// TwinCAT 3 PLC project PLC_CRIX_VAC
// Title: plc-crix-vac
// Company: SLAC - LCLS
// ProjectVersion: 0.0.0
// ProgramVersion: 3.1.4022.7
// libraries:
//   LCLS General, * (SLAC)
//   LCLS Vacuum, * (SLAC - LCLS)
//   LCLSVacuumSerialDriverLib, * (SLAC - LCLS)
//   PMPS, * (SLAC - LCLS)
//   Tc2_SerialCom, * (Beckhoff Automation GmbH)
//   Tc2_Standard, * (Beckhoff Automation GmbH)
//   Tc2_System, * (Beckhoff Automation GmbH)
//   Tc3_Module, * (Beckhoff Automation GmbH)
// project tree:
//   / CommTask.TcTTO, PlcTask.TcTTO
//   DUTs/ E_STATES.TcDUT
//   GVLs/ GVL_ADS_Devices.TcGVL, GVL_Chamber_Gauges.TcGVL, GVL_Chamber_Valves.TcGVL, GVL_COM.TcGVL, GVL_COM_VLS.TcGVL, GVL_LI3K2.TcGVL, GVL_Mech_Room.TcGVL, GVL_PLC_Interfaces.TcGVL, GVL_PMPS.TcGVL, GVL_Pumps.TcGVL, GVL_Recirculation.TcGVL, GVL_Vars.TcGVL, GVL_VLS.TcGVL
//   POUs/ FB_ChemRIXS_Turbo_ILK.TcPOU, F_TurboGateValve_Protection_ILK_Turbo_OFF_OK_NO_GPI_READ.TcPOU, MAIN.TcPOU, PRG_ADS_Gauges.TcPOU, PRG_ADS_Interfaces.TcPOU, PRG_Chamber_Gauges.TcPOU, PRG_Chamber_Pumps.TcPOU, PRG_Chamber_Valves.TcPOU, PRG_Com.TcPOU, PRG_COM_VLS.TcPOU, PRG_LI3K2.TcPOU, PRG_Mechanical_Room.TcPOU, PRG_MPS.TcPOU, PRG_RCC.TcPOU, PRG_VLS_Turbo.TcPOU, PRG_VLS_VACUUM.TcPOU, PRG_VLS_WINDOW.TcPOU
// real-time tasks:
//   TASK PlcTask: cycle T#10ms, priority 20, ADS port 350
//   TASK CommTask: cycle T#10ms, priority 21, ADS port 351
// I/O:
//   DEVICE Device 1 (EtherCAT), AmsNetId 172.21.140.47.2.1
//     Term 1 (EK1200) [EK1200-5000 EtherCAT Power supply (2A E-Bus)]
//       Term 47 (EL6070) [EL6070 1Ch. Licensing-Terminal]
//       Term 2 (EK1122) [EK1122 2 port EtherCAT junction]
//         Hoffman Box Vac EK1 (EK1100) [EK1100 EtherCAT Coupler (2A E-Bus)]
//           E1 (EL2794)
//           E2 (EL1088) [EL1088 8Ch. Dig. Input 24V, 3ms, negative]
//           E4 (EL6002) [EL6002 Interface 2Ch. (RS232)]
//           E5 (EL6022) [EL6022 Interface 2Ch. (RS422/485)]
//           E6 (EL6022) [EL6022 Interface 2Ch. (RS422/485)]
//           E7 (EL9410)
//           E8 (EL3174) [EL3174 4Ch. Ana. Input +/-10V Diff., +/-20mA SingleEnded, 16 Bit]
//           E11 (EL3174) [EL3174 4Ch. Ana. Input +/-10V Diff., +/-20mA SingleEnded, 16 Bit]
//           E14 (EL3174) [EL3174 4Ch. Ana. Input +/-10V Diff., +/-20mA SingleEnded, 16 Bit]
//           E17 (EL2624)
//           E18 (EL9505)
//           E19 (EL1124) [EL1124 4Ch. Dig. Input 5V, 10µs, Sensor Power]
//           E20 (EL9410) [EL9410 E-Bus Power Supplier  (Diagnostics)]
//           E21 (EL2004)
//           E22 (EL1004) [EL1004 4Ch. Dig. Input 24V, 3ms]
//           E23 (EL1004)
//           E24 (EL2004) [EL2004 4Ch. Dig. Output 24V, 0.5A]
//           E25 (EL1004)
//           E26 (EL2004) [EL2004 4Ch. Dig. Output 24V, 0.5A]
//           E27 (EL1004) [EL1004 4Ch. Dig. Input 24V, 3ms]
//           E28 (EL2004)
//           E29 (EL1004) [EL1004 4Ch. Dig. Input 24V, 3ms]
//           E30 (EL2004)
//           E31 (EL1004)
//           E32 (EL9410) [EL9410 E-Bus Power Supplier  (Diagnostics)]
//           E33 (EL1004) [EL1004 4Ch. Dig. Input 24V, 3ms]
//           E34 (EL2004) [EL2004 4Ch. Dig. Output 24V, 0.5A]
//           E35 (EL1004) [EL1004 4Ch. Dig. Input 24V, 3ms]
//           E36 (EL2004)
//           E37 (EL1004)
//           E38 (EL1004) [EL1004 4Ch. Dig. Input 24V, 3ms]
//           E39 (EL2004) [EL2004 4Ch. Dig. Output 24V, 0.5A]
//           E40 (EL1004)
//           E41 (EL1004) [EL1004 4Ch. Dig. Input 24V, 3ms]
//           E42 (EL1004) [EL1004 4Ch. Dig. Input 24V, 3ms]
//           E43 (EL2794) [EL2794 4Ch. Dig. Output 24V AC/DC, 2A, short-circuit-proof]
//           E44 (EL1088) [EL1088 8Ch. Dig. Input 24V, 3ms, negative]
//           E46 (EL1004) [EL1004 4Ch. Dig. Input 24V, 3ms]
//           E47 (EL2004) [EL2004 4Ch. Dig. Output 24V, 0.5A]
//           E48 (EL9410) [EL9410 E-Bus Power Supplier  (Diagnostics)]
//           E49 (EL1004) [EL1004 4Ch. Dig. Input 24V, 3ms]
//           E50 (EL2004) [EL2004 4Ch. Dig. Output 24V, 0.5A]
//           E51 (EL4134) [EL4134 4Ch. Ana. Output -10/+10V, 16bit]
//           VLS_RCC (EK1122) [EK1122 2 port EtherCAT junction]
//             VLS_EP1 (EP6002-0002)
//             VLS_EP2 (EP2338-0001)
//             VLS_EP3 (EP2339-0021) [EP2339-0021 16 Ch. Dig. Input/Output 24V, 0,5A, M8]
//             VLS_EP4 (EP2624-0002) [EP2624-0002 4Ch. Relay Output, NO (125V AC / 30V DC)]
//             VLS_EP5 (EP3174-0002)
//             RCC_EK0 (EK1100) [EK1100 EtherCAT Coupler (2A E-Bus)]
//               RCC_E1 (EL1004) [EL1004 4Ch. Dig. Input 24V, 3ms]
//               RCC_E2 (EL2004) [EL2004 4Ch. Dig. Output 24V, 0.5A]
//               RCC_E3 (EL1004)
//               RCC_E4 (EL1004) [EL1004 4Ch. Dig. Input 24V, 3ms]
//               RCC_E5 (EL2004) [EL2004 4Ch. Dig. Output 24V, 0.5A]
//               RCC_E6 (EL1004) [EL1004 4Ch. Dig. Input 24V, 3ms]
//               RCC_E7 (EL3314) [EL3314 4Ch. Ana. Input Thermocouple (TC)]
//               RCC_E8 (EL2794) [EL2794 4Ch. Dig. Output 24V AC/DC, 2A, short-circuit-proof]
//               RCC_E9 (EL9505) [EL9505 Power supply terminal 5V]
//               RCC_E10 (EL1124)
//               Term 143 (EL3174-0002) [EL3174-0002 4Ch. Ana. Input +/-10V, +/-20mA 16 Bit, Isolated Channels]
//               RCC_E11 (EL9011)
//             RCC_GPI (901P)
//           Term 145 (EK1122) [EK1122 2 port EtherCAT junction]
//             SVLS_PR01 E0 (EK1100) [EK1100 EtherCAT Coupler (2A E-Bus)]
//               SVLS_PR01 E1 (EL6070) [EL6070 1Ch. Licensing-Terminal]
//               SVLS_PR01 E2 (EL1004) [EL1004 4Ch. Dig. Input 24V, 3ms]
//               SVLS_PR01 E3 (EL2794) [EL2794 4Ch. Dig. Output 24V AC/DC, 2A, short-circuit-proof]
//               SVLS_PR01 E4 (EL6021) [EL6021 Interface (RS422/485)]
//               SVLS_PR01 E5 (EL1004) [EL1004 4Ch. Dig. Input 24V, 3ms]
//               SVLS_PR01 E6 (EL2004) [EL2004 4Ch. Dig. Output 24V, 0.5A]
//               SVLS_PR01 E9 (EL3174-0002) [EL3174-0002 4Ch. Ana. Input +/-10V, +/-20mA 16 Bit, Isolated Channels]
//               SVLS_PR01 E10 (EL9505) [EL9505 Power supply terminal 5V]
//               SVLS_PR01 E11 (EL1124) [EL1124 4Ch. Dig. Input 5V, 10µs, Sensor Power]
//               SVLS_PR01 E12 (EL6695) [EL6695 EtherCAT Bridge terminal (Primary)]
//               SVLS_PR01 E13 (EL9011) [EL9011 End Terminal]
//           E53 (EL9011)
//         Mech Room Vac EK1 (EK1101) [EK1101 EtherCAT Coupler (2A E-Bus, ID switch)]
//           Term 45 (EL2794) [EL2794 4Ch. Dig. Output 24V AC/DC, 2A, short-circuit-proof]
//           Term 83 (EL1088) [EL1088 8Ch. Dig. Input 24V, 3ms, negative]
//           Term 92 (EL3174) [EL3174 4Ch. Ana. Input +/-10V Diff., +/-20mA SingleEnded, 16 Bit]
//           Term 93 (EL1004) [EL1004 4Ch. Dig. Input 24V, 3ms]
//           Term 94 (EL2004) [EL2004 4Ch. Dig. Output 24V, 0.5A]
//           Term 153 (EL2212) [EL2212 2Ch. dig. output with overexcitation (24V DC, 2.5A, 10A Peak)]
//           Term 96 (EL9011) [EL9011 End Terminal]
//       Term 95 (EL6695) [EL6695 EtherCAT Bridge terminal (Primary)]
//       Term 113 (EK1521-0010) [EK1521-0010 1 port EtherCAT junction (FX-SingleMode)]
//         Term 154 (EK1501-0010) [EK1501-0010 EtherCAT Coupler (2A E-Bus, FX-SingleMode, ID switch)]
//           PMPS_FFO [EL2202 2Ch. Dig. Output 24V, 0.5A]
//           PMPS_PRE [EL6695 EtherCAT Bridge terminal (Primary)]
//           Term 159 (EL9011)
// variable links:
//   PLC_CRIX_VAC Instance <-> Device 1 (EtherCAT)/Term 1 (EK1200)/Term 113 (EK1521-0010)/Term 154 (EK1501-0010)/PMPS_FFO
//     PlcTask Outputs/GVL_PMPS.g_FastFaultOutput1.q_xFastFaultOut <-> Channel 1/Output
//   PLC_CRIX_VAC Instance <-> Device 1 (EtherCAT)/Term 1 (EK1200)/Term 113 (EK1521-0010)/Term 154 (EK1501-0010)/PMPS_PRE
//     PlcTask Inputs/PRG_MPS.fbArbiterIO.i_stCurrentBP <-> IO Inputs/CurrentBP
//     PlcTask Inputs/PRG_MPS.fbArbiterIO.xTxPDO_state <-> SYNC Inputs/TxPDO state
//     PlcTask Inputs/PRG_MPS.fbArbiterIO.xTxPDO_toggle <-> SYNC Inputs/TxPDO toggle
//     PlcTask Outputs/PRG_MPS.fbArbiterIO.q_stRequestedBP <-> IO Outputs/RequestedBP
//   PLC_CRIX_VAC Instance <-> Device 1 (EtherCAT)/Term 1 (EK1200)/Term 2 (EK1122)/Hoffman Box Vac EK1 (EK1100)/E11 (EL3174)
//     PlcTask Inputs/GVL_Chamber_Gauges.CRYO_GCP_01.i_iPRESS_R <-> AI Standard Channel 2/Value
//     PlcTask Inputs/GVL_Chamber_Gauges.CRYO_GCP_02.i_iPRESS_R <-> AI Standard Channel 1/Value
//     PlcTask Inputs/GVL_Chamber_Gauges.ROUGH_GPI_01.i_iPRESS_R <-> AI Standard Channel 4/Value
//     PlcTask Inputs/GVL_Chamber_Gauges.SDS_GCP_01.i_iPRESS_R <-> AI Standard Channel 3/Value
//   PLC_CRIX_VAC Instance <-> Device 1 (EtherCAT)/Term 1 (EK1200)/Term 2 (EK1122)/Hoffman Box Vac EK1 (EK1100)/E14 (EL3174)
//     PlcTask Inputs/GVL_Chamber_Gauges.TC_GCC_01.i_iPRESS_R <-> AI Standard Channel 1/Value
//   PLC_CRIX_VAC Instance <-> Device 1 (EtherCAT)/Term 1 (EK1200)/Term 2 (EK1122)/Hoffman Box Vac EK1 (EK1100)/E17 (EL2624)
//     PlcTask Outputs/GVL_Chamber_Gauges.TC_GCC_01.q_xHV_DIS <-> Channel 1/Output
//   PLC_CRIX_VAC Instance <-> Device 1 (EtherCAT)/Term 1 (EK1200)/Term 2 (EK1122)/Hoffman Box Vac EK1 (EK1100)/E19 (EL1124)
//     PlcTask Inputs/GVL_Chamber_Gauges.TC_GCC_01.i_xDisc_Active <-> Channel 2/Input
//     PlcTask Inputs/GVL_Chamber_Gauges.TC_GCC_01.i_xHV_ON <-> Channel 1/Input
//   PLC_CRIX_VAC Instance <-> Device 1 (EtherCAT)/Term 1 (EK1200)/Term 2 (EK1122)/Hoffman Box Vac EK1 (EK1100)/E21 (EL2004)
//     PlcTask Outputs/GVL_Chamber_Valves.TC_VRC_01.q_xOPN_DO <-> Channel 1/Output
//     PlcTask Outputs/GVL_Chamber_Valves.TC_VRC_02.q_xOPN_DO <-> Channel 2/Output
//     PlcTask Outputs/GVL_Chamber_Valves.TC_VRC_03.q_xOPN_DO <-> Channel 3/Output
//     PlcTask Outputs/GVL_Chamber_Valves.VLS_VRC_01.q_xOPN_DO <-> Channel 4/Output
//   PLC_CRIX_VAC Instance <-> Device 1 (EtherCAT)/Term 1 (EK1200)/Term 2 (EK1122)/Hoffman Box Vac EK1 (EK1100)/E22 (EL1004)
//     PlcTask Inputs/GVL_Chamber_Valves.TC_VRC_01.i_xClsLS <-> Channel 2/Input
//     PlcTask Inputs/GVL_Chamber_Valves.TC_VRC_02.i_xClsLS <-> Channel 4/Input
//     PlcTask Inputs/GVL_Chamber_Valves.TC_VRC_01.i_xOpnLS <-> Channel 1/Input
//     PlcTask Inputs/GVL_Chamber_Valves.TC_VRC_02.i_xOpnLS <-> Channel 3/Input
//   PLC_CRIX_VAC Instance <-> Device 1 (EtherCAT)/Term 1 (EK1200)/Term 2 (EK1122)/Hoffman Box Vac EK1 (EK1100)/E23 (EL1004)
//     PlcTask Inputs/GVL_Chamber_Valves.TC_VRC_03.i_xClsLS <-> Channel 2/Input
//     PlcTask Inputs/GVL_Chamber_Valves.TC_VRC_03.i_xOpnLS <-> Channel 1/Input
//     PlcTask Inputs/GVL_Chamber_Valves.VLS_VRC_01.i_xClsLS <-> Channel 4/Input
//     PlcTask Inputs/GVL_Chamber_Valves.VLS_VRC_01.i_xOpnLS <-> Channel 3/Input
//   PLC_CRIX_VAC Instance <-> Device 1 (EtherCAT)/Term 1 (EK1200)/Term 2 (EK1122)/Hoffman Box Vac EK1 (EK1100)/E24 (EL2004)
//     PlcTask Outputs/GVL_Chamber_Valves.MAIN_VGC_01.q_xOPN_DO <-> Channel 3/Output
//     PlcTask Outputs/GVL_Chamber_Valves.SDS_VRC_01.q_xOPN_DO <-> Channel 1/Output
//     PlcTask Outputs/GVL_Chamber_Valves.SDS_VRC_03.q_xOPN_DO <-> Channel 2/Output
//   PLC_CRIX_VAC Instance <-> Device 1 (EtherCAT)/Term 1 (EK1200)/Term 2 (EK1122)/Hoffman Box Vac EK1 (EK1100)/E25 (EL1004)
//     PlcTask Inputs/GVL_Chamber_Valves.SDS_VRC_01.i_xClsLS <-> Channel 2/Input
//     PlcTask Inputs/GVL_Chamber_Valves.SDS_VRC_03.i_xClsLS <-> Channel 4/Input
//     PlcTask Inputs/GVL_Chamber_Valves.SDS_VRC_01.i_xOpnLS <-> Channel 1/Input
//     PlcTask Inputs/GVL_Chamber_Valves.SDS_VRC_03.i_xOpnLS <-> Channel 3/Input
//   PLC_CRIX_VAC Instance <-> Device 1 (EtherCAT)/Term 1 (EK1200)/Term 2 (EK1122)/Hoffman Box Vac EK1 (EK1100)/E26 (EL2004)
//     PlcTask Outputs/GVL_Chamber_Valves.CRYO_VGC_01.q_xCLS_DO <-> Channel 3/Output
//     PlcTask Outputs/GVL_Chamber_Valves.CRYO_VGC_01.q_xOPN_DO <-> Channel 2/Output
//     PlcTask Outputs/GVL_Chamber_Valves.CRYO_VGC_02.q_xOPN_DO <-> Channel 4/Output
//     PlcTask Outputs/GVL_Chamber_Valves.MAIN_VGC_02.q_xOPN_DO <-> Channel 1/Output
//   PLC_CRIX_VAC Instance <-> Device 1 (EtherCAT)/Term 1 (EK1200)/Term 2 (EK1122)/Hoffman Box Vac EK1 (EK1100)/E27 (EL1004)
//     PlcTask Inputs/GVL_Chamber_Valves.MAIN_VGC_01.i_xClsLS <-> Channel 2/Input
//     PlcTask Inputs/GVL_Chamber_Valves.MAIN_VGC_01.i_xOpnLS <-> Channel 1/Input
//   PLC_CRIX_VAC Instance <-> Device 1 (EtherCAT)/Term 1 (EK1200)/Term 2 (EK1122)/Hoffman Box Vac EK1 (EK1100)/E28 (EL2004)
//     PlcTask Outputs/GVL_Chamber_Valves.CRYO_VGC_02.q_xCLS_DO <-> Channel 1/Output
//     PlcTask Outputs/GVL_Chamber_Valves.CRYO_VRC_01.q_xOPN_DO <-> Channel 2/Output
//     PlcTask Outputs/GVL_Chamber_Valves.CRYO_VRC_02.q_xOPN_DO <-> Channel 3/Output
//     PlcTask Outputs/GVL_Chamber_Valves.SDS_VGC_01.q_xOPN_DO <-> Channel 4/Output
//   PLC_CRIX_VAC Instance <-> Device 1 (EtherCAT)/Term 1 (EK1200)/Term 2 (EK1122)/Hoffman Box Vac EK1 (EK1100)/E29 (EL1004)
//     PlcTask Inputs/GVL_Chamber_Valves.MAIN_VGC_02.i_xClsLS <-> Channel 1/Input
//     PlcTask Inputs/GVL_Chamber_Valves.MAIN_VGC_02.i_xOpnLS <-> Channel 2/Input
//   PLC_CRIX_VAC Instance <-> Device 1 (EtherCAT)/Term 1 (EK1200)/Term 2 (EK1122)/Hoffman Box Vac EK1 (EK1100)/E30 (EL2004)
//     PlcTask Outputs/GVL_Chamber_Valves.SDS_VGC_01.q_xCLS_DO <-> Channel 1/Output
//     PlcTask Outputs/GVL_Chamber_Valves.SDS_VRC_02.q_xOPN_DO <-> Channel 2/Output
//   PLC_CRIX_VAC Instance <-> Device 1 (EtherCAT)/Term 1 (EK1200)/Term 2 (EK1122)/Hoffman Box Vac EK1 (EK1100)/E31 (EL1004)
//     PlcTask Inputs/GVL_Chamber_Valves.CRYO_VGC_01.i_xClsLS <-> Channel 2/Input
//     PlcTask Inputs/GVL_Chamber_Valves.CRYO_VGC_01.i_xOpnLS <-> Channel 1/Input
//     PlcTask Inputs/GVL_Chamber_Valves.CRYO_VRC_01.i_xClsLS <-> Channel 4/Input
//     PlcTask Inputs/GVL_Chamber_Valves.CRYO_VRC_01.i_xOpnLS <-> Channel 3/Input
//   PLC_CRIX_VAC Instance <-> Device 1 (EtherCAT)/Term 1 (EK1200)/Term 2 (EK1122)/Hoffman Box Vac EK1 (EK1100)/E33 (EL1004)
//     PlcTask Inputs/GVL_Chamber_Valves.CRYO_VGC_02.i_xClsLS <-> Channel 2/Input
//     PlcTask Inputs/GVL_Chamber_Valves.CRYO_VGC_02.i_xOpnLS <-> Channel 1/Input
//     PlcTask Inputs/GVL_Chamber_Valves.CRYO_VRC_02.i_xClsLS <-> Channel 4/Input
//     PlcTask Inputs/GVL_Chamber_Valves.CRYO_VRC_02.i_xOpnLS <-> Channel 3/Input
//   PLC_CRIX_VAC Instance <-> Device 1 (EtherCAT)/Term 1 (EK1200)/Term 2 (EK1122)/Hoffman Box Vac EK1 (EK1100)/E35 (EL1004)
//     PlcTask Inputs/GVL_Chamber_Valves.SDS_VGC_01.i_xClsLS <-> Channel 2/Input
//     PlcTask Inputs/GVL_Chamber_Valves.SDS_VGC_01.i_xOpnLS <-> Channel 1/Input
//   PLC_CRIX_VAC Instance <-> Device 1 (EtherCAT)/Term 1 (EK1200)/Term 2 (EK1122)/Hoffman Box Vac EK1 (EK1100)/E37 (EL1004)
//     PlcTask Inputs/GVL_Chamber_Valves.SDS_VRC_02.i_xClsLS <-> Channel 2/Input
//     PlcTask Inputs/GVL_Chamber_Valves.SDS_VRC_02.i_xOpnLS <-> Channel 1/Input
//   PLC_CRIX_VAC Instance <-> Device 1 (EtherCAT)/Term 1 (EK1200)/Term 2 (EK1122)/Hoffman Box Vac EK1 (EK1100)/E39 (EL2004)
//     PlcTask Outputs/GVL_Chamber_Valves.CRIX_SVLS_VRC_01.q_xOPN_DO <-> Channel 3/Output
//     PlcTask Outputs/GVL_Chamber_Valves.SDS_VVC_01.q_xOPN_DO <-> Channel 1/Output
//     PlcTask Outputs/GVL_Chamber_Valves.SDS_VVC_02.q_xOPN_DO <-> Channel 2/Output
//   PLC_CRIX_VAC Instance <-> Device 1 (EtherCAT)/Term 1 (EK1200)/Term 2 (EK1122)/Hoffman Box Vac EK1 (EK1100)/E40 (EL1004)
//     PlcTask Inputs/GVL_Chamber_Valves.SDS_VVC_01.i_xClsLS <-> Channel 3/Input
//     PlcTask Inputs/GVL_Chamber_Valves.SDS_VVC_02.i_xClsLS <-> Channel 4/Input
//   PLC_CRIX_VAC Instance <-> Device 1 (EtherCAT)/Term 1 (EK1200)/Term 2 (EK1122)/Hoffman Box Vac EK1 (EK1100)/E41 (EL1004)
//     PlcTask Inputs/GVL_Chamber_Valves.CRIX_SVLS_VRC_01.i_xClsLS <-> Channel 2/Input
//     PlcTask Inputs/GVL_Chamber_Valves.CRIX_SVLS_VRC_01.i_xOpnLS <-> Channel 1/Input
//   PLC_CRIX_VAC Instance <-> Device 1 (EtherCAT)/Term 1 (EK1200)/Term 2 (EK1122)/Hoffman Box Vac EK1 (EK1100)/E42 (EL1004)
//     PlcTask Inputs/GVL_Pumps.TC_PTM_01.i_xAtSpd <-> Channel 4/Input
//     PlcTask Inputs/GVL_Pumps.TC_PTM_02.i_xAtSpd <-> Channel 2/Input
//     PlcTask Inputs/GVL_Pumps.TC_PTM_01.i_xFaultNC <-> Channel 3/Input
//     PlcTask Inputs/GVL_Pumps.TC_PTM_02.i_xFaultNC <-> Channel 1/Input
//   PLC_CRIX_VAC Instance <-> Device 1 (EtherCAT)/Term 1 (EK1200)/Term 2 (EK1122)/Hoffman Box Vac EK1 (EK1100)/E43 (EL2794)
//     PlcTask Outputs/GVL_Pumps.TC_PTM_01.q_RunDO <-> Channel 4/Output
//     PlcTask Outputs/GVL_Pumps.TC_PTM_02.q_RunDO <-> Channel 3/Output
//   PLC_CRIX_VAC Instance <-> Device 1 (EtherCAT)/Term 1 (EK1200)/Term 2 (EK1122)/Hoffman Box Vac EK1 (EK1100)/E46 (EL1004)
//     PlcTask Inputs/GVL_Pumps.TC_PTM_03.i_xAtSpd <-> Channel 1/Input
//     PlcTask Inputs/GVL_Pumps.TC_PTM_03.i_xFaultNC <-> Channel 3/Input
//     PlcTask Inputs/GVL_Pumps.TC_PTM_03.i_xRemote <-> Channel 2/Input
//   PLC_CRIX_VAC Instance <-> Device 1 (EtherCAT)/Term 1 (EK1200)/Term 2 (EK1122)/Hoffman Box Vac EK1 (EK1100)/E47 (EL2004)
//     PlcTask Outputs/GVL_Pumps.TC_PTM_03.q_PumpingStation <-> Channel 3/Output
//     PlcTask Outputs/GVL_Pumps.TC_PTM_03.q_RunDO <-> Channel 1/Output
//     PlcTask Outputs/GVL_Pumps.TC_PTM_03.q_xRemote <-> Channel 2/Output
//   PLC_CRIX_VAC Instance <-> Device 1 (EtherCAT)/Term 1 (EK1200)/Term 2 (EK1122)/Hoffman Box Vac EK1 (EK1100)/E49 (EL1004)
//     PlcTask Inputs/GVL_Pumps.SDS_PTM_01.i_xAtSpd <-> Channel 1/Input
//     PlcTask Inputs/GVL_Pumps.SDS_PTM_01.i_xFaultNC <-> Channel 3/Input
//     PlcTask Inputs/GVL_Pumps.SDS_PTM_01.i_xRemote <-> Channel 2/Input
//   PLC_CRIX_VAC Instance <-> Device 1 (EtherCAT)/Term 1 (EK1200)/Term 2 (EK1122)/Hoffman Box Vac EK1 (EK1100)/E5 (EL6022)
//     PlcTask Inputs/GVL_COM.K2S17_E5_CH1_stComIn/D[0] <-> COM Inputs Channel 1/Data In 0
//     PlcTask Inputs/GVL_COM.K2S17_E5_CH1_stComIn/D[10] <-> COM Inputs Channel 1/Data In 10
//     PlcTask Inputs/GVL_COM.K2S17_E5_CH1_stComIn/D[11] <-> COM Inputs Channel 1/Data In 11
//     PlcTask Inputs/GVL_COM.K2S17_E5_CH1_stComIn/D[12] <-> COM Inputs Channel 1/Data In 12
//     PlcTask Inputs/GVL_COM.K2S17_E5_CH1_stComIn/D[13] <-> COM Inputs Channel 1/Data In 13
//     PlcTask Inputs/GVL_COM.K2S17_E5_CH1_stComIn/D[14] <-> COM Inputs Channel 1/Data In 14
//     PlcTask Inputs/GVL_COM.K2S17_E5_CH1_stComIn/D[15] <-> COM Inputs Channel 1/Data In 15
//     PlcTask Inputs/GVL_COM.K2S17_E5_CH1_stComIn/D[16] <-> COM Inputs Channel 1/Data In 16
//     PlcTask Inputs/GVL_COM.K2S17_E5_CH1_stComIn/D[17] <-> COM Inputs Channel 1/Data In 17
//     PlcTask Inputs/GVL_COM.K2S17_E5_CH1_stComIn/D[18] <-> COM Inputs Channel 1/Data In 18
//     PlcTask Inputs/GVL_COM.K2S17_E5_CH1_stComIn/D[19] <-> COM Inputs Channel 1/Data In 19
//     PlcTask Inputs/GVL_COM.K2S17_E5_CH1_stComIn/D[1] <-> COM Inputs Channel 1/Data In 1
//     PlcTask Inputs/GVL_COM.K2S17_E5_CH1_stComIn/D[20] <-> COM Inputs Channel 1/Data In 20
//     PlcTask Inputs/GVL_COM.K2S17_E5_CH1_stComIn/D[21] <-> COM Inputs Channel 1/Data In 21
//     PlcTask Inputs/GVL_COM.K2S17_E5_CH1_stComIn/D[2] <-> COM Inputs Channel 1/Data In 2
//     PlcTask Inputs/GVL_COM.K2S17_E5_CH1_stComIn/D[3] <-> COM Inputs Channel 1/Data In 3
//     PlcTask Inputs/GVL_COM.K2S17_E5_CH1_stComIn/D[4] <-> COM Inputs Channel 1/Data In 4
//     PlcTask Inputs/GVL_COM.K2S17_E5_CH1_stComIn/D[5] <-> COM Inputs Channel 1/Data In 5
//     PlcTask Inputs/GVL_COM.K2S17_E5_CH1_stComIn/D[6] <-> COM Inputs Channel 1/Data In 6
//     PlcTask Inputs/GVL_COM.K2S17_E5_CH1_stComIn/D[7] <-> COM Inputs Channel 1/Data In 7
//     PlcTask Inputs/GVL_COM.K2S17_E5_CH1_stComIn/D[8] <-> COM Inputs Channel 1/Data In 8
//     PlcTask Inputs/GVL_COM.K2S17_E5_CH1_stComIn/D[9] <-> COM Inputs Channel 1/Data In 9
//     PlcTask Inputs/GVL_COM.K2S17_E5_CH2_stComIn/D[0] <-> COM Inputs Channel 2/Data In 0
//     PlcTask Inputs/GVL_COM.K2S17_E5_CH2_stComIn/D[10] <-> COM Inputs Channel 2/Data In 10
//     PlcTask Inputs/GVL_COM.K2S17_E5_CH2_stComIn/D[11] <-> COM Inputs Channel 2/Data In 11
//     PlcTask Inputs/GVL_COM.K2S17_E5_CH2_stComIn/D[12] <-> COM Inputs Channel 2/Data In 12
//     PlcTask Inputs/GVL_COM.K2S17_E5_CH2_stComIn/D[13] <-> COM Inputs Channel 2/Data In 13
//     PlcTask Inputs/GVL_COM.K2S17_E5_CH2_stComIn/D[14] <-> COM Inputs Channel 2/Data In 14
//     PlcTask Inputs/GVL_COM.K2S17_E5_CH2_stComIn/D[15] <-> COM Inputs Channel 2/Data In 15
//     PlcTask Inputs/GVL_COM.K2S17_E5_CH2_stComIn/D[16] <-> COM Inputs Channel 2/Data In 16
//     PlcTask Inputs/GVL_COM.K2S17_E5_CH2_stComIn/D[17] <-> COM Inputs Channel 2/Data In 17
//     PlcTask Inputs/GVL_COM.K2S17_E5_CH2_stComIn/D[18] <-> COM Inputs Channel 2/Data In 18
//     PlcTask Inputs/GVL_COM.K2S17_E5_CH2_stComIn/D[19] <-> COM Inputs Channel 2/Data In 19
//     PlcTask Inputs/GVL_COM.K2S17_E5_CH2_stComIn/D[1] <-> COM Inputs Channel 2/Data In 1
//     PlcTask Inputs/GVL_COM.K2S17_E5_CH2_stComIn/D[20] <-> COM Inputs Channel 2/Data In 20
//     PlcTask Inputs/GVL_COM.K2S17_E5_CH2_stComIn/D[21] <-> COM Inputs Channel 2/Data In 21
//     PlcTask Inputs/GVL_COM.K2S17_E5_CH2_stComIn/D[2] <-> COM Inputs Channel 2/Data In 2
//     PlcTask Inputs/GVL_COM.K2S17_E5_CH2_stComIn/D[3] <-> COM Inputs Channel 2/Data In 3
//     PlcTask Inputs/GVL_COM.K2S17_E5_CH2_stComIn/D[4] <-> COM Inputs Channel 2/Data In 4
//     PlcTask Inputs/GVL_COM.K2S17_E5_CH2_stComIn/D[5] <-> COM Inputs Channel 2/Data In 5
//     PlcTask Inputs/GVL_COM.K2S17_E5_CH2_stComIn/D[6] <-> COM Inputs Channel 2/Data In 6
//     PlcTask Inputs/GVL_COM.K2S17_E5_CH2_stComIn/D[7] <-> COM Inputs Channel 2/Data In 7
//     PlcTask Inputs/GVL_COM.K2S17_E5_CH2_stComIn/D[8] <-> COM Inputs Channel 2/Data In 8
//     PlcTask Inputs/GVL_COM.K2S17_E5_CH2_stComIn/D[9] <-> COM Inputs Channel 2/Data In 9
//     PlcTask Inputs/GVL_COM.K2S17_E5_CH1_stComIn/Status <-> COM Inputs Channel 1/Status
//     PlcTask Inputs/GVL_COM.K2S17_E5_CH2_stComIn/Status <-> COM Inputs Channel 2/Status
//     PlcTask Outputs/GVL_COM.K2S17_E5_CH1_stComOut/Ctrl <-> COM Outputs Channel 1/Ctrl
//     PlcTask Outputs/GVL_COM.K2S17_E5_CH2_stComOut/Ctrl <-> COM Outputs Channel 2/Ctrl
//     PlcTask Outputs/GVL_COM.K2S17_E5_CH1_stComOut/D[0] <-> COM Outputs Channel 1/Data Out 0
//     PlcTask Outputs/GVL_COM.K2S17_E5_CH1_stComOut/D[10] <-> COM Outputs Channel 1/Data Out 10
//     PlcTask Outputs/GVL_COM.K2S17_E5_CH1_stComOut/D[11] <-> COM Outputs Channel 1/Data Out 11
//     PlcTask Outputs/GVL_COM.K2S17_E5_CH1_stComOut/D[12] <-> COM Outputs Channel 1/Data Out 12
//     PlcTask Outputs/GVL_COM.K2S17_E5_CH1_stComOut/D[13] <-> COM Outputs Channel 1/Data Out 13
//     PlcTask Outputs/GVL_COM.K2S17_E5_CH1_stComOut/D[14] <-> COM Outputs Channel 1/Data Out 14
//     PlcTask Outputs/GVL_COM.K2S17_E5_CH1_stComOut/D[15] <-> COM Outputs Channel 1/Data Out 15
//     PlcTask Outputs/GVL_COM.K2S17_E5_CH1_stComOut/D[16] <-> COM Outputs Channel 1/Data Out 16
//     PlcTask Outputs/GVL_COM.K2S17_E5_CH1_stComOut/D[17] <-> COM Outputs Channel 1/Data Out 17
//     PlcTask Outputs/GVL_COM.K2S17_E5_CH1_stComOut/D[18] <-> COM Outputs Channel 1/Data Out 18
//     PlcTask Outputs/GVL_COM.K2S17_E5_CH1_stComOut/D[19] <-> COM Outputs Channel 1/Data Out 19
//     PlcTask Outputs/GVL_COM.K2S17_E5_CH1_stComOut/D[1] <-> COM Outputs Channel 1/Data Out 1
//     PlcTask Outputs/GVL_COM.K2S17_E5_CH1_stComOut/D[20] <-> COM Outputs Channel 1/Data Out 20
//     PlcTask Outputs/GVL_COM.K2S17_E5_CH1_stComOut/D[21] <-> COM Outputs Channel 1/Data Out 21
//     PlcTask Outputs/GVL_COM.K2S17_E5_CH1_stComOut/D[2] <-> COM Outputs Channel 1/Data Out 2
//     PlcTask Outputs/GVL_COM.K2S17_E5_CH1_stComOut/D[3] <-> COM Outputs Channel 1/Data Out 3
//     PlcTask Outputs/GVL_COM.K2S17_E5_CH1_stComOut/D[4] <-> COM Outputs Channel 1/Data Out 4
//     PlcTask Outputs/GVL_COM.K2S17_E5_CH1_stComOut/D[5] <-> COM Outputs Channel 1/Data Out 5
//     PlcTask Outputs/GVL_COM.K2S17_E5_CH1_stComOut/D[6] <-> COM Outputs Channel 1/Data Out 6
//     PlcTask Outputs/GVL_COM.K2S17_E5_CH1_stComOut/D[7] <-> COM Outputs Channel 1/Data Out 7
//     PlcTask Outputs/GVL_COM.K2S17_E5_CH1_stComOut/D[8] <-> COM Outputs Channel 1/Data Out 8
//     PlcTask Outputs/GVL_COM.K2S17_E5_CH1_stComOut/D[9] <-> COM Outputs Channel 1/Data Out 9
//     PlcTask Outputs/GVL_COM.K2S17_E5_CH2_stComOut/D[0] <-> COM Outputs Channel 2/Data Out 0
//     PlcTask Outputs/GVL_COM.K2S17_E5_CH2_stComOut/D[10] <-> COM Outputs Channel 2/Data Out 10
//     PlcTask Outputs/GVL_COM.K2S17_E5_CH2_stComOut/D[11] <-> COM Outputs Channel 2/Data Out 11
//     PlcTask Outputs/GVL_COM.K2S17_E5_CH2_stComOut/D[12] <-> COM Outputs Channel 2/Data Out 12
//     PlcTask Outputs/GVL_COM.K2S17_E5_CH2_stComOut/D[13] <-> COM Outputs Channel 2/Data Out 13
//     PlcTask Outputs/GVL_COM.K2S17_E5_CH2_stComOut/D[14] <-> COM Outputs Channel 2/Data Out 14
//     PlcTask Outputs/GVL_COM.K2S17_E5_CH2_stComOut/D[15] <-> COM Outputs Channel 2/Data Out 15
//     PlcTask Outputs/GVL_COM.K2S17_E5_CH2_stComOut/D[16] <-> COM Outputs Channel 2/Data Out 16
//     PlcTask Outputs/GVL_COM.K2S17_E5_CH2_stComOut/D[17] <-> COM Outputs Channel 2/Data Out 17
//     PlcTask Outputs/GVL_COM.K2S17_E5_CH2_stComOut/D[18] <-> COM Outputs Channel 2/Data Out 18
//     PlcTask Outputs/GVL_COM.K2S17_E5_CH2_stComOut/D[19] <-> COM Outputs Channel 2/Data Out 19
//     PlcTask Outputs/GVL_COM.K2S17_E5_CH2_stComOut/D[1] <-> COM Outputs Channel 2/Data Out 1
//     PlcTask Outputs/GVL_COM.K2S17_E5_CH2_stComOut/D[20] <-> COM Outputs Channel 2/Data Out 20
//     PlcTask Outputs/GVL_COM.K2S17_E5_CH2_stComOut/D[21] <-> COM Outputs Channel 2/Data Out 21
//     PlcTask Outputs/GVL_COM.K2S17_E5_CH2_stComOut/D[2] <-> COM Outputs Channel 2/Data Out 2
//     PlcTask Outputs/GVL_COM.K2S17_E5_CH2_stComOut/D[3] <-> COM Outputs Channel 2/Data Out 3
//     PlcTask Outputs/GVL_COM.K2S17_E5_CH2_stComOut/D[4] <-> COM Outputs Channel 2/Data Out 4
//     PlcTask Outputs/GVL_COM.K2S17_E5_CH2_stComOut/D[5] <-> COM Outputs Channel 2/Data Out 5
//     PlcTask Outputs/GVL_COM.K2S17_E5_CH2_stComOut/D[6] <-> COM Outputs Channel 2/Data Out 6
//     PlcTask Outputs/GVL_COM.K2S17_E5_CH2_stComOut/D[7] <-> COM Outputs Channel 2/Data Out 7
//     PlcTask Outputs/GVL_COM.K2S17_E5_CH2_stComOut/D[8] <-> COM Outputs Channel 2/Data Out 8
//     PlcTask Outputs/GVL_COM.K2S17_E5_CH2_stComOut/D[9] <-> COM Outputs Channel 2/Data Out 9
//   PLC_CRIX_VAC Instance <-> Device 1 (EtherCAT)/Term 1 (EK1200)/Term 2 (EK1122)/Hoffman Box Vac EK1 (EK1100)/E50 (EL2004)
//     PlcTask Outputs/GVL_Pumps.SDS_PTM_01.q_PumpingStation <-> Channel 3/Output
//     PlcTask Outputs/GVL_Pumps.SDS_PTM_01.q_RunDO <-> Channel 1/Output
//     PlcTask Outputs/GVL_Pumps.SDS_PTM_01.q_xRemote <-> Channel 2/Output
//   PLC_CRIX_VAC Instance <-> Device 1 (EtherCAT)/Term 1 (EK1200)/Term 2 (EK1122)/Hoffman Box Vac EK1 (EK1100)/E8 (EL3174)
//     PlcTask Inputs/GVL_Chamber_Gauges.CRYO_GPI_01.i_iPRESS_R <-> AI Standard Channel 3/Value
//     PlcTask Inputs/GVL_Chamber_Gauges.TC_GCP_01.i_iPRESS_R <-> AI Standard Channel 4/Value
//     PlcTask Inputs/GVL_Chamber_Gauges.TC_GPI_01.i_iPRESS_R <-> AI Standard Channel 2/Value
//   PLC_CRIX_VAC Instance <-> Device 1 (EtherCAT)/Term 1 (EK1200)/Term 2 (EK1122)/Hoffman Box Vac EK1 (EK1100)/Term 145 (EK1122)/SVLS_PR01 E0 (EK1100)/SVLS_PR01 E11 (EL1124)
//     PlcTask Inputs/GVL_Pumps.CRIX_SVLS_PIP_1.i_xError <-> Channel 2/Input
//     PlcTask Inputs/GVL_Pumps.CRIX_SVLS_PIP_1.i_xIP_ON <-> Channel 1/Input
//   PLC_CRIX_VAC Instance <-> Device 1 (EtherCAT)/Term 1 (EK1200)/Term 2 (EK1122)/Hoffman Box Vac EK1 (EK1100)/Term 145 (EK1122)/SVLS_PR01 E0 (EK1100)/SVLS_PR01 E2 (EL1004)
//     PlcTask Inputs/GVL_Pumps.CRIX_SVLS_PTM_01.i_xAtSpd <-> Channel 1/Input
//     PlcTask Inputs/GVL_Pumps.CRIX_SVLS_PTM_01.i_xFaultNC <-> Channel 2/Input
//   PLC_CRIX_VAC Instance <-> Device 1 (EtherCAT)/Term 1 (EK1200)/Term 2 (EK1122)/Hoffman Box Vac EK1 (EK1100)/Term 145 (EK1122)/SVLS_PR01 E0 (EK1100)/SVLS_PR01 E3 (EL2794)
//     PlcTask Outputs/GVL_Pumps.CRIX_SVLS_PIP_1.q_xHVEna_DO <-> Channel 3/Output
//     PlcTask Outputs/GVL_Pumps.CRIX_SVLS_PTM_01.q_RunDO <-> Channel 1/Output
//     PlcTask Outputs/GVL_Pumps.CRIX_SVLS_PTM_01.q_xReset <-> Channel 2/Output
//   PLC_CRIX_VAC Instance <-> Device 1 (EtherCAT)/Term 1 (EK1200)/Term 2 (EK1122)/Hoffman Box Vac EK1 (EK1100)/Term 145 (EK1122)/SVLS_PR01 E0 (EK1100)/SVLS_PR01 E4 (EL6021)
//     PlcTask Inputs/GVL_COM.CRIX_SVLS_stComIn/D[{0..21}] <-> COM TxPDO-Map Inputs/Data In {0..21}  (22 links)
//     PlcTask Inputs/GVL_COM.CRIX_SVLS_stComIn/Status <-> COM TxPDO-Map Inputs/Status
//     PlcTask Outputs/GVL_COM.CRIX_SVLS_stComOut/Ctrl <-> COM RxPDO-Map Outputs/Ctrl
//     PlcTask Outputs/GVL_COM.CRIX_SVLS_stComOut/D[{0..21}] <-> COM RxPDO-Map Outputs/Data Out {0..21}  (22 links)
//   PLC_CRIX_VAC Instance <-> Device 1 (EtherCAT)/Term 1 (EK1200)/Term 2 (EK1122)/Hoffman Box Vac EK1 (EK1100)/Term 145 (EK1122)/SVLS_PR01 E0 (EK1100)/SVLS_PR01 E5 (EL1004)
//     PlcTask Inputs/GVL_Chamber_Valves.CRIX_SVLS_VWC_01.i_xClsLS <-> Channel 2/Input
//     PlcTask Inputs/GVL_Chamber_Valves.CRIX_SVLS_VWC_01.i_xOpnLS <-> Channel 1/Input
//   PLC_CRIX_VAC Instance <-> Device 1 (EtherCAT)/Term 1 (EK1200)/Term 2 (EK1122)/Hoffman Box Vac EK1 (EK1100)/Term 145 (EK1122)/SVLS_PR01 E0 (EK1100)/SVLS_PR01 E6 (EL2004)
//     PlcTask Outputs/GVL_Chamber_Valves.CRIX_SVLS_VWC_01.q_xCLS_DO <-> Channel 1/Output
//   PLC_CRIX_VAC Instance <-> Device 1 (EtherCAT)/Term 1 (EK1200)/Term 2 (EK1122)/Hoffman Box Vac EK1 (EK1100)/Term 145 (EK1122)/SVLS_PR01 E0 (EK1100)/SVLS_PR01 E9 (EL3174-0002)
//     PlcTask Inputs/GVL_Chamber_Gauges.CRIX_SVLS_GCP_01.i_iPRESS_R <-> AI Standard Channel 1/Value
//     PlcTask Inputs/GVL_Chamber_Gauges.CRIX_SVLS_GCP_02.i_iPRESS_R <-> AI Standard Channel 2/Value
//     PlcTask Inputs/GVL_Pumps.CRIX_SVLS_PIP_1.i_iPRESS <-> AI Standard Channel 1/Value
//   PLC_CRIX_VAC Instance <-> Device 1 (EtherCAT)/Term 1 (EK1200)/Term 2 (EK1122)/Hoffman Box Vac EK1 (EK1100)/VLS_RCC (EK1122)/RCC_EK0 (EK1100)/RCC_E1 (EL1004)
//     PlcTask Inputs/GVL_Recirculation.RCC_VRC_01.i_xClsLS <-> Channel 1/Input
//     PlcTask Inputs/GVL_Recirculation.RCC_VRC_02.i_xClsLS <-> Channel 2/Input
//     PlcTask Inputs/GVL_Recirculation.RCC_VRC_03.i_xClsLS <-> Channel 3/Input
//     PlcTask Inputs/GVL_Recirculation.RCC_VRC_02.i_xOpnLS <-> Channel 4/Input
//   PLC_CRIX_VAC Instance <-> Device 1 (EtherCAT)/Term 1 (EK1200)/Term 2 (EK1122)/Hoffman Box Vac EK1 (EK1100)/VLS_RCC (EK1122)/RCC_EK0 (EK1100)/RCC_E2 (EL2004)
//     PlcTask Outputs/GVL_Recirculation.RCC_VRC_01.q_xOPN_DO <-> Channel 1/Output
//     PlcTask Outputs/GVL_Recirculation.RCC_VRC_02.q_xOPN_DO <-> Channel 2/Output
//     PlcTask Outputs/GVL_Recirculation.RCC_VRC_03.q_xOPN_DO <-> Channel 3/Output
//     PlcTask Outputs/GVL_Recirculation.RCC_VRC_04.q_xOPN_DO <-> Channel 4/Output
//   PLC_CRIX_VAC Instance <-> Device 1 (EtherCAT)/Term 1 (EK1200)/Term 2 (EK1122)/Hoffman Box Vac EK1 (EK1100)/VLS_RCC (EK1122)/RCC_EK0 (EK1100)/RCC_E3 (EL1004)
//     PlcTask Inputs/GVL_Recirculation.RCC_VRC_04.i_xClsLS <-> Channel 1/Input
//   PLC_CRIX_VAC Instance <-> Device 1 (EtherCAT)/Term 1 (EK1200)/Term 2 (EK1122)/Hoffman Box Vac EK1 (EK1100)/VLS_RCC (EK1122)/RCC_EK0 (EK1100)/RCC_E7 (EL3314)
//     PlcTask Inputs/GVL_Recirculation.RCC_STC_01.bError <-> TC Inputs Channel 3/Status/Error
//     PlcTask Inputs/GVL_Recirculation.RCC_STC_02.bError <-> TC Inputs Channel 4/Status/Error
//     PlcTask Inputs/GVL_Recirculation.RCC_STC_01.bOverrange <-> TC Inputs Channel 3/Status/Overrange
//     PlcTask Inputs/GVL_Recirculation.RCC_STC_02.bOverrange <-> TC Inputs Channel 4/Status/Overrange
//     PlcTask Inputs/GVL_Recirculation.RCC_STC_01.bUnderrange <-> TC Inputs Channel 3/Status/Underrange
//     PlcTask Inputs/GVL_Recirculation.RCC_STC_02.bUnderrange <-> TC Inputs Channel 4/Status/Underrange
//     PlcTask Inputs/GVL_Recirculation.RCC_STC_01.iRaw <-> TC Inputs Channel 3/Value
//     PlcTask Inputs/GVL_Recirculation.RCC_STC_02.iRaw <-> TC Inputs Channel 4/Value
//   PLC_CRIX_VAC Instance <-> Device 1 (EtherCAT)/Term 1 (EK1200)/Term 2 (EK1122)/Hoffman Box Vac EK1 (EK1100)/VLS_RCC (EK1122)/RCC_GPI (901P)
//     PlcTask Inputs/GVL_Recirculation.RCC_GCP_01.bWcstate <-> WcState/WcState
//     PlcTask Inputs/GVL_Recirculation.RCC_GCP_01.i_iPRESS_R <-> TXPDO Combined/Combination Gauge Active Value
//     PlcTask Inputs/GVL_Recirculation.RCC_GCP_01.xOverrange <-> TXPDO Combined/Combination Gauge Overrange Exceeded
//     PlcTask Inputs/GVL_Recirculation.RCC_GCP_01.xPress_OK <-> TXPDO Combined/Combination Gauge Reading Valid
//     PlcTask Inputs/GVL_Recirculation.RCC_GCP_01.xUnderrange <-> TXPDO Combined/Combination Gauge Underrange Exceeded
//   PLC_CRIX_VAC Instance <-> Device 1 (EtherCAT)/Term 1 (EK1200)/Term 2 (EK1122)/Hoffman Box Vac EK1 (EK1100)/VLS_RCC (EK1122)/VLS_EP1 (EP6002-0002)
//     PlcTask Inputs/GVL_COM_VLS.VLS_EP1_CH1_stComIn/D[{0..21}] <-> COM TxPDO-Map Inputs Channel 1/Data In {0..21}  (22 links)
//     PlcTask Inputs/GVL_COM_VLS.VLS_EP1_CH1_stComIn/Status <-> COM TxPDO-Map Inputs Channel 1/Status
//     PlcTask Outputs/GVL_COM_VLS.VLS_EP1_CH1_stComOut/Ctrl <-> COM RxPDO-Map Outputs Channel 1/Ctrl
//     PlcTask Outputs/GVL_COM_VLS.VLS_EP1_CH1_stComOut/D[{0..21}] <-> COM RxPDO-Map Outputs Channel 1/Data Out {0..21}  (22 links)
//   PLC_CRIX_VAC Instance <-> Device 1 (EtherCAT)/Term 1 (EK1200)/Term 2 (EK1122)/Hoffman Box Vac EK1 (EK1100)/VLS_RCC (EK1122)/VLS_EP2 (EP2338-0001)
//     PlcTask Inputs/GVL_VLS.VLS_PTM_01.i_xAtSpd <-> Channel 1/Input
//     PlcTask Inputs/GVL_VLS.VLS_PTM_01.i_xFaultNC <-> Channel 2/Input
//   PLC_CRIX_VAC Instance <-> Device 1 (EtherCAT)/Term 1 (EK1200)/Term 2 (EK1122)/Hoffman Box Vac EK1 (EK1100)/VLS_RCC (EK1122)/VLS_EP3 (EP2339-0021)
//     PlcTask Inputs/GVL_VLS.VLS_VGC_01.i_xClsLS <-> Channel 7/Input
//     PlcTask Inputs/GVL_VLS.VLS_VGC_01.i_xOpnLS <-> Channel 6/Input
//     PlcTask Inputs/GVL_VLS.VLS_VWC_01.i_xClsLS <-> Channel 10/Input
//     PlcTask Inputs/GVL_VLS.VLS_VWC_01.i_xOpnLS <-> Channel 9/Input
//     PlcTask Outputs/GVL_VLS.VLS_VGC_01.q_xOPN_DO <-> Channel 21/Output
//     PlcTask Outputs/GVL_VLS.VLS_VWC_01.q_xCLS_DO <-> Channel 24/Output
//   PLC_CRIX_VAC Instance <-> Device 1 (EtherCAT)/Term 1 (EK1200)/Term 2 (EK1122)/Hoffman Box Vac EK1 (EK1100)/VLS_RCC (EK1122)/VLS_EP4 (EP2624-0002)
//     PlcTask Outputs/GVL_VLS.VLS_GCC_01.q_xHV_DIS <-> Channel 1/Output
//     PlcTask Outputs/GVL_VLS.VLS_PTM_01.q_RunDO <-> Channel 3/Output
//   PLC_CRIX_VAC Instance <-> Device 1 (EtherCAT)/Term 1 (EK1200)/Term 2 (EK1122)/Hoffman Box Vac EK1 (EK1100)/VLS_RCC (EK1122)/VLS_EP5 (EP3174-0002)
//     PlcTask Inputs/GVL_VLS.VLS_GCC_01.i_iPRESS_R <-> AI Standard Channel 2/Value
//     PlcTask Inputs/GVL_VLS.VLS_GPI_01.i_iPRESS_R <-> AI Standard Channel 1/Value
//     PlcTask Inputs/GVL_VLS.VLS_ROUGH_GPI.i_iPRESS_R <-> AI Standard Channel 3/Value
//   PLC_CRIX_VAC Instance <-> Device 1 (EtherCAT)/Term 1 (EK1200)/Term 2 (EK1122)/Mech Room Vac EK1 (EK1101)/Term 153 (EL2212)
//     PlcTask Outputs/GVL_Mech_Room.MECH_VVC_01.q_xOPN_DO <-> DOX Control Channel 2/Control/Output
//   PLC_CRIX_VAC Instance <-> Device 1 (EtherCAT)/Term 1 (EK1200)/Term 2 (EK1122)/Mech Room Vac EK1 (EK1101)/Term 45 (EL2794)
//     PlcTask Outputs/GVL_Mech_Room.MECH_PRO_01.q_xBPStart <-> Channel 2/Output
//     PlcTask Outputs/GVL_Mech_Room.MECH_PRO_01.q_xMPStart <-> Channel 1/Output
//   PLC_CRIX_VAC Instance <-> Device 1 (EtherCAT)/Term 1 (EK1200)/Term 2 (EK1122)/Mech Room Vac EK1 (EK1101)/Term 83 (EL1088)
//     PlcTask Inputs/GVL_Mech_Room.MECH_PRO_01.i_xAlarmOK <-> Channel 4/Input
//     PlcTask Inputs/GVL_Mech_Room.MECH_PRO_01.i_xBPStatus <-> Channel 2/Input
//     PlcTask Inputs/GVL_Mech_Room.MECH_PRO_01.i_xMPStatus <-> Channel 1/Input
//     PlcTask Inputs/GVL_Mech_Room.MECH_PRO_01.i_xRemote <-> Channel 5/Input
//     PlcTask Inputs/GVL_Mech_Room.MECH_PRO_01.i_xWarning <-> Channel 3/Input
//   PLC_CRIX_VAC Instance <-> Device 1 (EtherCAT)/Term 1 (EK1200)/Term 2 (EK1122)/Mech Room Vac EK1 (EK1101)/Term 92 (EL3174)
//     PlcTask Inputs/GVL_Mech_Room.MECH_GPI_01.i_iPRESS_R <-> AI Standard Channel 1/Value
//   PLC_CRIX_VAC Instance <-> Device 1 (EtherCAT)/Term 1 (EK1200)/Term 95 (EL6695)
//     PlcTask Inputs/GVL_PLC_Interfaces.xEcatBridge_External_device_not_connected <-> SYNC Inputs/External device not connected
//     PlcTask Inputs/GVL_PLC_Interfaces.xEcatBridge_TxPDO_state <-> SYNC Inputs/TxPDO state
//     PlcTask Inputs/GVL_PLC_Interfaces.xEcatBridge_WcState <-> WcState/WcState
//     PlcTask Inputs/GVL_PLC_Interfaces.xPTC_MOT_Y_10_IN <-> IO Inputs/bMOTY10_IN
//     PlcTask Inputs/GVL_PLC_Interfaces.xPTC_MOT_Y_11_IN <-> IO Inputs/bMOTY11_IN
//     PlcTask Inputs/GVL_PLC_Interfaces.xPTC_MOT_Y_10_OUT <-> IO Inputs/bMOTY10_OUT
//     PlcTask Inputs/GVL_PLC_Interfaces.xPTC_MOT_Y_11_OUT <-> IO Inputs/bMOTY11_OUT
//     PlcTask Inputs/GVL_PLC_Interfaces.xSDS_MOT_Z_18_IN <-> IO Inputs/xSDS_MOT_Z_18_IN
//     PlcTask Inputs/GVL_PLC_Interfaces.xSDS_MOT_Z_18_OUT <-> IO Inputs/xSDS_MOT_Z_18_OUT
//     PlcTask Outputs/GVL_PLC_Interfaces.bCRYO_VGC_01_CLS <-> IO Outputs/bCRYO_VGC_01_CLS
//     PlcTask Outputs/GVL_PLC_Interfaces.bCRYO_VGC_02_CLS <-> IO Outputs/bCRYO_VGC_02_CLS
//     PlcTask Outputs/GVL_PLC_Interfaces.bCRYO_VGC_01_OPN <-> IO Outputs/bCRYO_VGC_01_OPN
//     PlcTask Outputs/GVL_PLC_Interfaces.bCRYO_VGC_02_OPN <-> IO Outputs/bCRYO_VGC_02_OPN
//     PlcTask Outputs/GVL_PLC_Interfaces.bSDS_VGC_01_CLS <-> IO Outputs/bSDS_VGC_01_CLS
//     PlcTask Outputs/GVL_PLC_Interfaces.bSDS_VGC_01_OPN <-> IO Outputs/bSDS_VGC_01_OPN

CONFIGURATION PLC_CRIX_VAC
    RESOURCE PLC ON TwinCAT3
        TASK CommTask(INTERVAL := T#10ms, PRIORITY := 21);
        TASK PlcTask(INTERVAL := T#10ms, PRIORITY := 20);
        PROGRAM PRG_COM_VLS WITH CommTask : PRG_COM_VLS;
        PROGRAM MAIN WITH PlcTask : MAIN;
    END_RESOURCE
END_CONFIGURATION

// ---- DUTs/E_STATES.TcDUT
{attribute 'qualified_only'}
{attribute 'strict'}
TYPE E_STATES :
(
    INIT := 0,
    SETUP,
    OVERRIDE,
    READY,
    NOT_SAFE
);
END_TYPE

// ---- GVLs/GVL_ADS_Devices.TcGVL
//{attribute 'qualified_only'}
VAR_GLOBAL

 {attribute 'pytmc' :=' pv: TM2K2:GCC:01:reader '}
    TM2K2_GCC_01_reader : FB_TGCC_ADS;
 {attribute 'pytmc' :=' pv: AT3K2:GCC:01:reader '}
    AT3K2_GCC_01_reader : FB_TGCC_ADS;

END_VAR

// ---- GVLs/GVL_Chamber_Gauges.TcGVL
//{attribute 'qualified_only'}
VAR_GLOBAL
    (* Pirani & Cold Cathode*)

    {attribute 'pytmc' :=' pv: CRIXS:TC:GPI:01 '}
    {attribute 'TcLinkTo' := 	'.i_iPRESS_R	:=	TIID^Device 1 (EtherCAT)^Term 1 (EK1200)^Term 2 (EK1122)^Hoffman Box Vac EK1 (EK1100)^E8 (EL3174)^AI Standard Channel 2^Value '}
    TC_GPI_01 : FB_MKS275;

    stTC_GPI_01 : ST_VG;


    {attribute 'pytmc' :=' pv: CRIXS:CRYO:GPI:01 '}
    {attribute 'TcLinkTo' := 	'.i_iPRESS_R	:=	TIID^Device 1 (EtherCAT)^Term 1 (EK1200)^Term 2 (EK1122)^Hoffman Box Vac EK1 (EK1100)^E8 (EL3174)^AI Standard Channel 3^Value '}
    CRYO_GPI_01 : FB_MKS275;

    stCRYO_GPI_01 : ST_VG;


    {attribute 'pytmc' :=' pv: CRIXS:ROUGH:GPI:01 '}
    {attribute 'TcLinkTo' := 	'.i_iPRESS_R	:=	TIID^Device 1 (EtherCAT)^Term 1 (EK1200)^Term 2 (EK1122)^Hoffman Box Vac EK1 (EK1100)^E11 (EL3174)^AI Standard Channel 4^Value '}
    ROUGH_GPI_01 : FB_MKS275;

    stROUGH_GPI_01 : ST_VG;

    {attribute 'pytmc' :=' pv: CRIXS:TC:GCC:01 '}
    {attribute 'TcLinkTo' := 	'.i_iPRESS_R	:=	TIID^Device 1 (EtherCAT)^Term 1 (EK1200)^Term 2 (EK1122)^Hoffman Box Vac EK1 (EK1100)^E14 (EL3174)^AI Standard Channel 1^Value;
                                 .i_xHV_ON	    :=	TIID^Device 1 (EtherCAT)^Term 1 (EK1200)^Term 2 (EK1122)^Hoffman Box Vac EK1 (EK1100)^E19 (EL1124)^Channel 1^Input;
                                 .i_xDisc_Active:=	TIID^Device 1 (EtherCAT)^Term 1 (EK1200)^Term 2 (EK1122)^Hoffman Box Vac EK1 (EK1100)^E19 (EL1124)^Channel 2^Input;
                                 .q_xHV_DIS		:= 	TIID^Device 1 (EtherCAT)^Term 1 (EK1200)^Term 2 (EK1122)^Hoffman Box Vac EK1 (EK1100)^E17 (EL2624)^Channel 1^Output	'}
    TC_GCC_01 : FB_MKS500;

    stTC_GCC_01 : ST_VG;

    (* Micro Pirani combination gauges *)


    {attribute 'pytmc' :=' pv: CRIXS:CRYO:GCP:01 '}
    {attribute 'TcLinkTo' := 	'.i_iPRESS_R	:= TIID^Device 1 (EtherCAT)^Term 1 (EK1200)^Term 2 (EK1122)^Hoffman Box Vac EK1 (EK1100)^E11 (EL3174)^AI Standard Channel 2^Value '}
    CRYO_GCP_01 : FB_972;

    stCRYO_GCP_01 : ST_VG;

    {attribute 'pytmc' :=' pv: CRIXS:CRYO:GCP:02 '}
    {attribute 'TcLinkTo' := 	'.i_iPRESS_R	:= TIID^Device 1 (EtherCAT)^Term 1 (EK1200)^Term 2 (EK1122)^Hoffman Box Vac EK1 (EK1100)^E11 (EL3174)^AI Standard Channel 1^Value '}
    CRYO_GCP_02 : FB_972;

    stCRYO_GCP_02 : ST_VG;

    {attribute 'pytmc' :=' pv: CRIXS:SDS:GCP:01 '}
    {attribute 'TcLinkTo' := 	'.i_iPRESS_R	:= TIID^Device 1 (EtherCAT)^Term 1 (EK1200)^Term 2 (EK1122)^Hoffman Box Vac EK1 (EK1100)^E11 (EL3174)^AI Standard Channel 3^Value '}
    SDS_GCP_01 : FB_972;

    stSDS_GCP_01 : ST_VG;

    {attribute 'pytmc' :=' pv: CRIXS:TC:GCP:01 '}
    {attribute 'TcLinkTo' := 	'.i_iPRESS_R	:=	TIID^Device 1 (EtherCAT)^Term 1 (EK1200)^Term 2 (EK1122)^Hoffman Box Vac EK1 (EK1100)^E8 (EL3174)^AI Standard Channel 4^Value '}
    TC_GCP_01 : FB_972;

    stTC_GCP_01 : ST_VG;

    {attribute 'pytmc' :=' pv: CRIXS:SVLS:GCP:01 '}
    {attribute 'TcLinkTo' := 	'.i_iPRESS_R	:=	TIIB[SVLS_PR01 E9 (EL3174-0002)]^AI Standard Channel 1^Value '}
    CRIX_SVLS_GCP_01 : FB_972;

    stCRIX_SVLS_GCP_01 : ST_VG;

    {attribute 'pytmc' :=' pv: CRIXS:SVLS:GCP:02 '}
    {attribute 'TcLinkTo' := 	'.i_iPRESS_R	:=	TIIB[SVLS_PR01 E9 (EL3174-0002)]^AI Standard Channel 2^Value '}
    CRIX_SVLS_GCP_02 : FB_972;

    stCRIX_SVLS_GCP_02 : ST_VG;

END_VAR

// ---- GVLs/GVL_Chamber_Valves.TcGVL
//{attribute 'qualified_only'}
VAR_GLOBAL

    (* Roughing Manifold Valvese *)

    (*
    {attribute 'pytmc' :=' pv: CRIX:VGC:01 '}
    {attribute 'TcLinkTo' := 	'.i_xOpnLS	:=	TIID^Device 1 (EtherCAT)^Term 1 (EK1200)^Term 2 (EK1122)^Hoffman Box Vac EK1 (EK1100)^E41 (EL1004)^Channel 1^Input;
                                 .i_xClsLS	:=	TIID^Device 1 (EtherCAT)^Term 1 (EK1200)^Term 2 (EK1122)^Hoffman Box Vac EK1 (EK1100)^E41 (EL1004)^Channel 2^Input;
                                .q_xOPN_DO	:=	TIID^Device 1 (EtherCAT)^Term 1 (EK1200)^Term 2 (EK1122)^Hoffman Box Vac EK1 (EK1100)^E39 (EL2004)^Channel 3^Output'}
    CRIX_VGC_01 : FB_VRC;

    stCRIX_VGC_01 : ST_VRC;
    *)

    {attribute 'pytmc' :=' pv: CRIXS:TC:VRC:01 '}
    {attribute 'TcLinkTo' := 	'.i_xOpnLS	:=	TIID^Device 1 (EtherCAT)^Term 1 (EK1200)^Term 2 (EK1122)^Hoffman Box Vac EK1 (EK1100)^E22 (EL1004)^Channel 1^Input;
                                 .i_xClsLS	:=	TIID^Device 1 (EtherCAT)^Term 1 (EK1200)^Term 2 (EK1122)^Hoffman Box Vac EK1 (EK1100)^E22 (EL1004)^Channel 2^Input;
                                .q_xOPN_DO	:=	TIID^Device 1 (EtherCAT)^Term 1 (EK1200)^Term 2 (EK1122)^Hoffman Box Vac EK1 (EK1100)^E21 (EL2004)^Channel 1^Output'}

    TC_VRC_01 : FB_VGC_2S;

    stTC_VRC_01 : ST_VGC_2S;

    {attribute 'pytmc' :=' pv: CRIXS:TC:VRC:02 '}
    {attribute 'TcLinkTo' := 	'.i_xOpnLS	:=	TIID^Device 1 (EtherCAT)^Term 1 (EK1200)^Term 2 (EK1122)^Hoffman Box Vac EK1 (EK1100)^E22 (EL1004)^Channel 3^Input;
                                 .i_xClsLS	:=	TIID^Device 1 (EtherCAT)^Term 1 (EK1200)^Term 2 (EK1122)^Hoffman Box Vac EK1 (EK1100)^E22 (EL1004)^Channel 4^Input;
                                .q_xOPN_DO	:=	TIID^Device 1 (EtherCAT)^Term 1 (EK1200)^Term 2 (EK1122)^Hoffman Box Vac EK1 (EK1100)^E21 (EL2004)^Channel 2^Output'}

    TC_VRC_02 : FB_VRC;

    stTC_VRC_02 : ST_VRC;

    {attribute 'pytmc' :=' pv: CRIXS:TC:VRC:03 '}
    {attribute 'TcLinkTo' := 	'.i_xOpnLS	:=	TIID^Device 1 (EtherCAT)^Term 1 (EK1200)^Term 2 (EK1122)^Hoffman Box Vac EK1 (EK1100)^E23 (EL1004)^Channel 1^Input;
                                 .i_xClsLS	:=	TIID^Device 1 (EtherCAT)^Term 1 (EK1200)^Term 2 (EK1122)^Hoffman Box Vac EK1 (EK1100)^E23 (EL1004)^Channel 2^Input;
                                .q_xOPN_DO	:=	TIID^Device 1 (EtherCAT)^Term 1 (EK1200)^Term 2 (EK1122)^Hoffman Box Vac EK1 (EK1100)^E21 (EL2004)^Channel 3^Output'}

    TC_VRC_03 : FB_VRC;
    stTC_VRC_03 : ST_VRC;


    {attribute 'pytmc' :=' pv: CRIXS:VLS:VRC:01 '}
    {attribute 'TcLinkTo' := 	'.i_xOpnLS	:=	TIID^Device 1 (EtherCAT)^Term 1 (EK1200)^Term 2 (EK1122)^Hoffman Box Vac EK1 (EK1100)^E23 (EL1004)^Channel 3^Input;
                                 .i_xClsLS	:=	TIID^Device 1 (EtherCAT)^Term 1 (EK1200)^Term 2 (EK1122)^Hoffman Box Vac EK1 (EK1100)^E23 (EL1004)^Channel 4^Input;
                                .q_xOPN_DO	:=	TIID^Device 1 (EtherCAT)^Term 1 (EK1200)^Term 2 (EK1122)^Hoffman Box Vac EK1 (EK1100)^E21 (EL2004)^Channel 4^Output'}

    VLS_VRC_01 : FB_VRC;

    stVLS_VRC_01 : ST_VRC;

    (*
    stCRIX_VGC_03 : ST_VRC;
    *)
    {attribute 'pytmc' :=' pv: CRIXS:SDS:VRC:03 '}
    {attribute 'TcLinkTo' := 	'.i_xOpnLS	:=	TIID^Device 1 (EtherCAT)^Term 1 (EK1200)^Term 2 (EK1122)^Hoffman Box Vac EK1 (EK1100)^E25 (EL1004)^Channel 3^Input;
                                 .i_xClsLS	:=	TIID^Device 1 (EtherCAT)^Term 1 (EK1200)^Term 2 (EK1122)^Hoffman Box Vac EK1 (EK1100)^E25 (EL1004)^Channel 4^Input;
                                .q_xOPN_DO	:=	TIID^Device 1 (EtherCAT)^Term 1 (EK1200)^Term 2 (EK1122)^Hoffman Box Vac EK1 (EK1100)^E24 (EL2004)^Channel 2^Output'}

    SDS_VRC_03 : FB_VRC;

    /// Entry and Exit Valves for Target Chamber
    {attribute 'pytmc' :=' pv: CRIXS:MAIN:VGC:01 '}
    {attribute 'TcLinkTo' := 	'.i_xOpnLS	:=	TIID^Device 1 (EtherCAT)^Term 1 (EK1200)^Term 2 (EK1122)^Hoffman Box Vac EK1 (EK1100)^E27 (EL1004)^Channel 1^Input;
                                 .i_xClsLS	:=	TIID^Device 1 (EtherCAT)^Term 1 (EK1200)^Term 2 (EK1122)^Hoffman Box Vac EK1 (EK1100)^E27 (EL1004)^Channel 2^Input;
                                .q_xOPN_DO	:=	TIID^Device 1 (EtherCAT)^Term 1 (EK1200)^Term 2 (EK1122)^Hoffman Box Vac EK1 (EK1100)^E24 (EL2004)^Channel 3^Output'}

    MAIN_VGC_01 : FB_VGC;

    {attribute 'pytmc' :=' pv: CRIXS:MAIN:VGC:02 '}
    {attribute 'TcLinkTo' := 	'.i_xOpnLS	:=	TIID^Device 1 (EtherCAT)^Term 1 (EK1200)^Term 2 (EK1122)^Hoffman Box Vac EK1 (EK1100)^E29 (EL1004)^Channel 2^Input;
                                 .i_xClsLS	:=	TIID^Device 1 (EtherCAT)^Term 1 (EK1200)^Term 2 (EK1122)^Hoffman Box Vac EK1 (EK1100)^E29 (EL1004)^Channel 1^Input;
                                 .q_xOPN_DO	:=	TIID^Device 1 (EtherCAT)^Term 1 (EK1200)^Term 2 (EK1122)^Hoffman Box Vac EK1 (EK1100)^E26 (EL2004)^Channel 1^Output'}
    MAIN_VGC_02 : FB_VGC;

    /// Cryopump Roughing and Double Action Valves
    {attribute 'pytmc' :=' pv: CRIXS:CRYO:VGC:01 '}
    {attribute 'TcLinkTo' := 	'.i_xOpnLS	:=	TIID^Device 1 (EtherCAT)^Term 1 (EK1200)^Term 2 (EK1122)^Hoffman Box Vac EK1 (EK1100)^E31 (EL1004)^Channel 1^Input;
                                 .i_xClsLS	:=	TIID^Device 1 (EtherCAT)^Term 1 (EK1200)^Term 2 (EK1122)^Hoffman Box Vac EK1 (EK1100)^E31 (EL1004)^Channel 2^Input;
                                .q_xOPN_DO	:=	TIID^Device 1 (EtherCAT)^Term 1 (EK1200)^Term 2 (EK1122)^Hoffman Box Vac EK1 (EK1100)^E26 (EL2004)^Channel 2^Output;
                                .q_xCLS_DO	:=	TIID^Device 1 (EtherCAT)^Term 1 (EK1200)^Term 2 (EK1122)^Hoffman Box Vac EK1 (EK1100)^E26 (EL2004)^Channel 3^Output'}


    CRYO_VGC_01 : FB_VRC_DA;

    {attribute 'pytmc' :=' pv: CRIXS:CRYO:VGC:02 '}

     {attribute 'TcLinkTo' := 	'.i_xOpnLS	:=	TIID^Device 1 (EtherCAT)^Term 1 (EK1200)^Term 2 (EK1122)^Hoffman Box Vac EK1 (EK1100)^E33 (EL1004)^Channel 1^Input;
                                 .i_xClsLS	:=	TIID^Device 1 (EtherCAT)^Term 1 (EK1200)^Term 2 (EK1122)^Hoffman Box Vac EK1 (EK1100)^E33 (EL1004)^Channel 2^Input;
                                .q_xOPN_DO	:=	TIID^Device 1 (EtherCAT)^Term 1 (EK1200)^Term 2 (EK1122)^Hoffman Box Vac EK1 (EK1100)^E26 (EL2004)^Channel 4^Output;
                                .q_xCLS_DO	:=	TIID^Device 1 (EtherCAT)^Term 1 (EK1200)^Term 2 (EK1122)^Hoffman Box Vac EK1 (EK1100)^E28 (EL2004)^Channel 1^Output'}

    CRYO_VGC_02 : FB_VRC_DA;


    {attribute 'pytmc' :=' pv: CRIXS:CRYO:VRC:01 '}

    {attribute 'TcLinkTo' := 	'.i_xOpnLS	:=	TIID^Device 1 (EtherCAT)^Term 1 (EK1200)^Term 2 (EK1122)^Hoffman Box Vac EK1 (EK1100)^E31 (EL1004)^Channel 3^Input;
                                 .i_xClsLS	:=	TIID^Device 1 (EtherCAT)^Term 1 (EK1200)^Term 2 (EK1122)^Hoffman Box Vac EK1 (EK1100)^E31 (EL1004)^Channel 4^Input;
                                 .q_xOPN_DO	:=	TIID^Device 1 (EtherCAT)^Term 1 (EK1200)^Term 2 (EK1122)^Hoffman Box Vac EK1 (EK1100)^E28 (EL2004)^Channel 2^Output'}
    CRYO_VRC_01 : FB_VRC;


    {attribute 'pytmc' :=' pv: CRIXS:CRYO:VRC:02 '}

    {attribute 'TcLinkTo' := 	'.i_xOpnLS	:=	TIID^Device 1 (EtherCAT)^Term 1 (EK1200)^Term 2 (EK1122)^Hoffman Box Vac EK1 (EK1100)^E33 (EL1004)^Channel 3^Input;
                                 .i_xClsLS	:=	TIID^Device 1 (EtherCAT)^Term 1 (EK1200)^Term 2 (EK1122)^Hoffman Box Vac EK1 (EK1100)^E33 (EL1004)^Channel 4^Input;
                                 .q_xOPN_DO	:=	TIID^Device 1 (EtherCAT)^Term 1 (EK1200)^Term 2 (EK1122)^Hoffman Box Vac EK1 (EK1100)^E28 (EL2004)^Channel 3^Output'}
    CRYO_VRC_02 : FB_VRC;


    /// SDS Valves
    {attribute 'pytmc' :=' pv: CRIXS:SDS:VGC:01 '}
    {attribute 'TcLinkTo' := 	'.i_xOpnLS	:=	TIID^Device 1 (EtherCAT)^Term 1 (EK1200)^Term 2 (EK1122)^Hoffman Box Vac EK1 (EK1100)^E35 (EL1004)^Channel 1^Input;
                                 .i_xClsLS	:=	TIID^Device 1 (EtherCAT)^Term 1 (EK1200)^Term 2 (EK1122)^Hoffman Box Vac EK1 (EK1100)^E35 (EL1004)^Channel 2^Input;
                                .q_xOPN_DO	:=	TIID^Device 1 (EtherCAT)^Term 1 (EK1200)^Term 2 (EK1122)^Hoffman Box Vac EK1 (EK1100)^E28 (EL2004)^Channel 4^Output;
                                .q_xCLS_DO	:=	TIID^Device 1 (EtherCAT)^Term 1 (EK1200)^Term 2 (EK1122)^Hoffman Box Vac EK1 (EK1100)^E30 (EL2004)^Channel 1^Output'}
    SDS_VGC_01 : FB_VRC_DA;

    {attribute 'pytmc' :=' pv: CRIXS:SDS:VRC:02 '}
    {attribute 'TcLinkTo' := 	'.i_xOpnLS	:=	TIID^Device 1 (EtherCAT)^Term 1 (EK1200)^Term 2 (EK1122)^Hoffman Box Vac EK1 (EK1100)^E37 (EL1004)^Channel 1^Input;
                                 .i_xClsLS	:=	TIID^Device 1 (EtherCAT)^Term 1 (EK1200)^Term 2 (EK1122)^Hoffman Box Vac EK1 (EK1100)^E37 (EL1004)^Channel 2^Input;
                                .q_xOPN_DO	:=	TIID^Device 1 (EtherCAT)^Term 1 (EK1200)^Term 2 (EK1122)^Hoffman Box Vac EK1 (EK1100)^E30 (EL2004)^Channel 2^Output'}

    SDS_VRC_02 : FB_VRC;

    stSDS_VRC_02 : ST_VRC;

    {attribute 'pytmc' :=' pv: CRIXS:SDS:VRC:01 '}
    {attribute 'TcLinkTo' := 	'.i_xOpnLS	:=	TIID^Device 1 (EtherCAT)^Term 1 (EK1200)^Term 2 (EK1122)^Hoffman Box Vac EK1 (EK1100)^E25 (EL1004)^Channel 1^Input;
                                 .i_xClsLS	:=	TIID^Device 1 (EtherCAT)^Term 1 (EK1200)^Term 2 (EK1122)^Hoffman Box Vac EK1 (EK1100)^E25 (EL1004)^Channel 2^Input;
                                .q_xOPN_DO	:=	TIID^Device 1 (EtherCAT)^Term 1 (EK1200)^Term 2 (EK1122)^Hoffman Box Vac EK1 (EK1100)^E24 (EL2004)^Channel 1^Output'}

    SDS_VRC_01 : FB_VRC;

    stSDS_VRC_01 : ST_VRC;

     // Vent Package Valves
    {attribute 'pytmc' :=' pv: CRIXS:SDS:VVC:01 '}
    {attribute 'TcLinkTo' := 	'.i_xClsLS	:=	TIID^Device 1 (EtherCAT)^Term 1 (EK1200)^Term 2 (EK1122)^Hoffman Box Vac EK1 (EK1100)^E40 (EL1004)^Channel 3^Input;
                                .q_xOPN_DO	:=	TIID^Device 1 (EtherCAT)^Term 1 (EK1200)^Term 2 (EK1122)^Hoffman Box Vac EK1 (EK1100)^E39 (EL2004)^Channel 1^Output'}
    SDS_VVC_01 : FB_VRC_NC_ClsLs;

    {attribute 'pytmc' :=' pv: CRIXS:SDS:VVC:02 '}
    {attribute 'TcLinkTo' := 	'.i_xClsLS	:=	TIID^Device 1 (EtherCAT)^Term 1 (EK1200)^Term 2 (EK1122)^Hoffman Box Vac EK1 (EK1100)^E40 (EL1004)^Channel 4^Input;
                                .q_xOPN_DO	:=	TIID^Device 1 (EtherCAT)^Term 1 (EK1200)^Term 2 (EK1122)^Hoffman Box Vac EK1 (EK1100)^E39 (EL2004)^Channel 2^Output'}
    SDS_VVC_02 : FB_VRC_NC_ClsLs;

    {attribute 'pytmc' :=' pv: CRIXS:SVLS:VWC:01 '}
    {attribute 'TcLinkTo' := 	'.i_xOpnLS	:=	TIIB[SVLS_PR01 E5 (EL1004)]^Channel 1^Input;
                                 .i_xClsLS	:=	TIIB[SVLS_PR01 E5 (EL1004)]^Channel 2^Input;
                                .q_xCLS_DO	:=	TIIB[SVLS_PR01 E6 (EL2004)]^Channel 1^Output'}

    CRIX_SVLS_VWC_01 : FB_VRC_NO;

    stCRIX_SVLS_VWC_01 : ST_VRC_NO;

    {attribute 'pytmc' :=' pv: CRIXS:SVLS:VRC:01 '}
    {attribute 'TcLinkTo' := 	'.i_xOpnLS	:=	TIID^Device 1 (EtherCAT)^Term 1 (EK1200)^Term 2 (EK1122)^Hoffman Box Vac EK1 (EK1100)^E41 (EL1004)^Channel 1^Input;
                                 .i_xClsLS	:=	TIID^Device 1 (EtherCAT)^Term 1 (EK1200)^Term 2 (EK1122)^Hoffman Box Vac EK1 (EK1100)^E41 (EL1004)^Channel 2^Input;
                                 .q_xOPN_DO	:=	TIID^Device 1 (EtherCAT)^Term 1 (EK1200)^Term 2 (EK1122)^Hoffman Box Vac EK1 (EK1100)^E39 (EL2004)^Channel 3^Output'}

    CRIX_SVLS_VRC_01 : FB_VRC;

    stCRIX_SVLS_VRC_01 : ST_VRC;

END_VAR

// ---- GVLs/GVL_COM.TcGVL
//{attribute 'qualified_only'}
VAR_GLOBAL
    // PTM-03 on CH2, PTM-04 on CH1
    K2S17_E5_CH2_SerialRXBuffer : ComBuffer;
    K2S17_E5_CH2_SerialTXBuffer : ComBuffer;

    // Serial Terminal
    K2S17_E5_CH2_fbSerialLineControl: SerialLineControl;

    //SERIAL IO K2S17_E5_CH2 (EL6022)
    {attribute	'TcLinkTo'	:=	'.Status:=TIID^Device 1 (EtherCAT)^Term 1 (EK1200)^Term 2 (EK1122)^Hoffman Box Vac EK1 (EK1100)^E5 (EL6022)^COM Inputs Channel 2^Status;
                                 .D[0]:=TIID^Device 1 (EtherCAT)^Term 1 (EK1200)^Term 2 (EK1122)^Hoffman Box Vac EK1 (EK1100)^E5 (EL6022)^COM Inputs Channel 2^Data In 0;
                                 .D[1]:=TIID^Device 1 (EtherCAT)^Term 1 (EK1200)^Term 2 (EK1122)^Hoffman Box Vac EK1 (EK1100)^E5 (EL6022)^COM Inputs Channel 2^Data In 1;
                                 .D[2]:=TIID^Device 1 (EtherCAT)^Term 1 (EK1200)^Term 2 (EK1122)^Hoffman Box Vac EK1 (EK1100)^E5 (EL6022)^COM Inputs Channel 2^Data In 2;
                                 .D[3]:=TIID^Device 1 (EtherCAT)^Term 1 (EK1200)^Term 2 (EK1122)^Hoffman Box Vac EK1 (EK1100)^E5 (EL6022)^COM Inputs Channel 2^Data In 3;
                                 .D[4]:=TIID^Device 1 (EtherCAT)^Term 1 (EK1200)^Term 2 (EK1122)^Hoffman Box Vac EK1 (EK1100)^E5 (EL6022)^COM Inputs Channel 2^Data In 4;
                                 .D[5]:=TIID^Device 1 (EtherCAT)^Term 1 (EK1200)^Term 2 (EK1122)^Hoffman Box Vac EK1 (EK1100)^E5 (EL6022)^COM Inputs Channel 2^Data In 5;
                                 .D[6]:=TIID^Device 1 (EtherCAT)^Term 1 (EK1200)^Term 2 (EK1122)^Hoffman Box Vac EK1 (EK1100)^E5 (EL6022)^COM Inputs Channel 2^Data In 6;
                                 .D[7]:=TIID^Device 1 (EtherCAT)^Term 1 (EK1200)^Term 2 (EK1122)^Hoffman Box Vac EK1 (EK1100)^E5 (EL6022)^COM Inputs Channel 2^Data In 7;
                                 .D[8]:=TIID^Device 1 (EtherCAT)^Term 1 (EK1200)^Term 2 (EK1122)^Hoffman Box Vac EK1 (EK1100)^E5 (EL6022)^COM Inputs Channel 2^Data In 8;
                                 .D[9]:=TIID^Device 1 (EtherCAT)^Term 1 (EK1200)^Term 2 (EK1122)^Hoffman Box Vac EK1 (EK1100)^E5 (EL6022)^COM Inputs Channel 2^Data In 9;
                                 .D[10]:=TIID^Device 1 (EtherCAT)^Term 1 (EK1200)^Term 2 (EK1122)^Hoffman Box Vac EK1 (EK1100)^E5 (EL6022)^COM Inputs Channel 2^Data In 10;
                                 .D[11]:=TIID^Device 1 (EtherCAT)^Term 1 (EK1200)^Term 2 (EK1122)^Hoffman Box Vac EK1 (EK1100)^E5 (EL6022)^COM Inputs Channel 2^Data In 11;
                                 .D[12]:=TIID^Device 1 (EtherCAT)^Term 1 (EK1200)^Term 2 (EK1122)^Hoffman Box Vac EK1 (EK1100)^E5 (EL6022)^COM Inputs Channel 2^Data In 12;
                                 .D[13]:=TIID^Device 1 (EtherCAT)^Term 1 (EK1200)^Term 2 (EK1122)^Hoffman Box Vac EK1 (EK1100)^E5 (EL6022)^COM Inputs Channel 2^Data In 13;
                                 .D[14]:=TIID^Device 1 (EtherCAT)^Term 1 (EK1200)^Term 2 (EK1122)^Hoffman Box Vac EK1 (EK1100)^E5 (EL6022)^COM Inputs Channel 2^Data In 14;
                                 .D[15]:=TIID^Device 1 (EtherCAT)^Term 1 (EK1200)^Term 2 (EK1122)^Hoffman Box Vac EK1 (EK1100)^E5 (EL6022)^COM Inputs Channel 2^Data In 15;
                                 .D[16]:=TIID^Device 1 (EtherCAT)^Term 1 (EK1200)^Term 2 (EK1122)^Hoffman Box Vac EK1 (EK1100)^E5 (EL6022)^COM Inputs Channel 2^Data In 16;
                                 .D[17]:=TIID^Device 1 (EtherCAT)^Term 1 (EK1200)^Term 2 (EK1122)^Hoffman Box Vac EK1 (EK1100)^E5 (EL6022)^COM Inputs Channel 2^Data In 17;
                                 .D[18]:=TIID^Device 1 (EtherCAT)^Term 1 (EK1200)^Term 2 (EK1122)^Hoffman Box Vac EK1 (EK1100)^E5 (EL6022)^COM Inputs Channel 2^Data In 18;
                                 .D[19]:=TIID^Device 1 (EtherCAT)^Term 1 (EK1200)^Term 2 (EK1122)^Hoffman Box Vac EK1 (EK1100)^E5 (EL6022)^COM Inputs Channel 2^Data In 19;
                                 .D[20]:=TIID^Device 1 (EtherCAT)^Term 1 (EK1200)^Term 2 (EK1122)^Hoffman Box Vac EK1 (EK1100)^E5 (EL6022)^COM Inputs Channel 2^Data In 20;
                                 .D[21]:=TIID^Device 1 (EtherCAT)^Term 1 (EK1200)^Term 2 (EK1122)^Hoffman Box Vac EK1 (EK1100)^E5 (EL6022)^COM Inputs Channel 2^Data In 21
    '}
    K2S17_E5_CH2_stComIn		AT %I*	:	EL6inData22B;
    {attribute	'TcLinkTo'	:=	'.Ctrl:=TIID^Device 1 (EtherCAT)^Term 1 (EK1200)^Term 2 (EK1122)^Hoffman Box Vac EK1 (EK1100)^E5 (EL6022)^COM Outputs Channel 2^Ctrl;
                                 .D[0]:=TIID^Device 1 (EtherCAT)^Term 1 (EK1200)^Term 2 (EK1122)^Hoffman Box Vac EK1 (EK1100)^E5 (EL6022)^COM Outputs Channel 2^Data Out 0;
                                 .D[1]:=TIID^Device 1 (EtherCAT)^Term 1 (EK1200)^Term 2 (EK1122)^Hoffman Box Vac EK1 (EK1100)^E5 (EL6022)^COM Outputs Channel 2^Data Out 1;
                                 .D[2]:=TIID^Device 1 (EtherCAT)^Term 1 (EK1200)^Term 2 (EK1122)^Hoffman Box Vac EK1 (EK1100)^E5 (EL6022)^COM Outputs Channel 2^Data Out 2;
                                 .D[3]:=TIID^Device 1 (EtherCAT)^Term 1 (EK1200)^Term 2 (EK1122)^Hoffman Box Vac EK1 (EK1100)^E5 (EL6022)^COM Outputs Channel 2^Data Out 3;
                                 .D[4]:=TIID^Device 1 (EtherCAT)^Term 1 (EK1200)^Term 2 (EK1122)^Hoffman Box Vac EK1 (EK1100)^E5 (EL6022)^COM Outputs Channel 2^Data Out 4;
                                 .D[5]:=TIID^Device 1 (EtherCAT)^Term 1 (EK1200)^Term 2 (EK1122)^Hoffman Box Vac EK1 (EK1100)^E5 (EL6022)^COM Outputs Channel 2^Data Out 5;
                                 .D[6]:=TIID^Device 1 (EtherCAT)^Term 1 (EK1200)^Term 2 (EK1122)^Hoffman Box Vac EK1 (EK1100)^E5 (EL6022)^COM Outputs Channel 2^Data Out 6;
                                 .D[7]:=TIID^Device 1 (EtherCAT)^Term 1 (EK1200)^Term 2 (EK1122)^Hoffman Box Vac EK1 (EK1100)^E5 (EL6022)^COM Outputs Channel 2^Data Out 7;
                                 .D[8]:=TIID^Device 1 (EtherCAT)^Term 1 (EK1200)^Term 2 (EK1122)^Hoffman Box Vac EK1 (EK1100)^E5 (EL6022)^COM Outputs Channel 2^Data Out 8;
                                 .D[9]:=TIID^Device 1 (EtherCAT)^Term 1 (EK1200)^Term 2 (EK1122)^Hoffman Box Vac EK1 (EK1100)^E5 (EL6022)^COM Outputs Channel 2^Data Out 9;
                                 .D[10]:=TIID^Device 1 (EtherCAT)^Term 1 (EK1200)^Term 2 (EK1122)^Hoffman Box Vac EK1 (EK1100)^E5 (EL6022)^COM Outputs Channel 2^Data Out 10;
                                 .D[11]:=TIID^Device 1 (EtherCAT)^Term 1 (EK1200)^Term 2 (EK1122)^Hoffman Box Vac EK1 (EK1100)^E5 (EL6022)^COM Outputs Channel 2^Data Out 11;
                                 .D[12]:=TIID^Device 1 (EtherCAT)^Term 1 (EK1200)^Term 2 (EK1122)^Hoffman Box Vac EK1 (EK1100)^E5 (EL6022)^COM Outputs Channel 2^Data Out 12;
                                 .D[13]:=TIID^Device 1 (EtherCAT)^Term 1 (EK1200)^Term 2 (EK1122)^Hoffman Box Vac EK1 (EK1100)^E5 (EL6022)^COM Outputs Channel 2^Data Out 13;
                                 .D[14]:=TIID^Device 1 (EtherCAT)^Term 1 (EK1200)^Term 2 (EK1122)^Hoffman Box Vac EK1 (EK1100)^E5 (EL6022)^COM Outputs Channel 2^Data Out 14;
                                 .D[15]:=TIID^Device 1 (EtherCAT)^Term 1 (EK1200)^Term 2 (EK1122)^Hoffman Box Vac EK1 (EK1100)^E5 (EL6022)^COM Outputs Channel 2^Data Out 15;
                                 .D[16]:=TIID^Device 1 (EtherCAT)^Term 1 (EK1200)^Term 2 (EK1122)^Hoffman Box Vac EK1 (EK1100)^E5 (EL6022)^COM Outputs Channel 2^Data Out 16;
                                 .D[17]:=TIID^Device 1 (EtherCAT)^Term 1 (EK1200)^Term 2 (EK1122)^Hoffman Box Vac EK1 (EK1100)^E5 (EL6022)^COM Outputs Channel 2^Data Out 17;
                                 .D[18]:=TIID^Device 1 (EtherCAT)^Term 1 (EK1200)^Term 2 (EK1122)^Hoffman Box Vac EK1 (EK1100)^E5 (EL6022)^COM Outputs Channel 2^Data Out 18;
                                 .D[19]:=TIID^Device 1 (EtherCAT)^Term 1 (EK1200)^Term 2 (EK1122)^Hoffman Box Vac EK1 (EK1100)^E5 (EL6022)^COM Outputs Channel 2^Data Out 19;
                                 .D[20]:=TIID^Device 1 (EtherCAT)^Term 1 (EK1200)^Term 2 (EK1122)^Hoffman Box Vac EK1 (EK1100)^E5 (EL6022)^COM Outputs Channel 2^Data Out 20;
                                 .D[21]:=TIID^Device 1 (EtherCAT)^Term 1 (EK1200)^Term 2 (EK1122)^Hoffman Box Vac EK1 (EK1100)^E5 (EL6022)^COM Outputs Channel 2^Data Out 21
    '}
    K2S17_E5_CH2_stComOut		AT %Q*	:	EL6outData22B;



    // PTM-04 on CH1
    K2S17_E5_CH1_SerialRXBuffer : ComBuffer;
    K2S17_E5_CH1_SerialTXBuffer : ComBuffer;

    // Serial Terminal
    K2S17_E5_CH1_fbSerialLineControl: SerialLineControl;

    //SERIAL IO K2S17_E5_CH1 (EL6022)
    {attribute	'TcLinkTo'	:=	'.Status:=TIID^Device 1 (EtherCAT)^Term 1 (EK1200)^Term 2 (EK1122)^Hoffman Box Vac EK1 (EK1100)^E5 (EL6022)^COM Inputs Channel 1^Status;
                                 .D[0]:=TIID^Device 1 (EtherCAT)^Term 1 (EK1200)^Term 2 (EK1122)^Hoffman Box Vac EK1 (EK1100)^E5 (EL6022)^COM Inputs Channel 1^Data In 0;
                                 .D[1]:=TIID^Device 1 (EtherCAT)^Term 1 (EK1200)^Term 2 (EK1122)^Hoffman Box Vac EK1 (EK1100)^E5 (EL6022)^COM Inputs Channel 1^Data In 1;
                                 .D[2]:=TIID^Device 1 (EtherCAT)^Term 1 (EK1200)^Term 2 (EK1122)^Hoffman Box Vac EK1 (EK1100)^E5 (EL6022)^COM Inputs Channel 1^Data In 2;
                                 .D[3]:=TIID^Device 1 (EtherCAT)^Term 1 (EK1200)^Term 2 (EK1122)^Hoffman Box Vac EK1 (EK1100)^E5 (EL6022)^COM Inputs Channel 1^Data In 3;
                                 .D[4]:=TIID^Device 1 (EtherCAT)^Term 1 (EK1200)^Term 2 (EK1122)^Hoffman Box Vac EK1 (EK1100)^E5 (EL6022)^COM Inputs Channel 1^Data In 4;
                                 .D[5]:=TIID^Device 1 (EtherCAT)^Term 1 (EK1200)^Term 2 (EK1122)^Hoffman Box Vac EK1 (EK1100)^E5 (EL6022)^COM Inputs Channel 1^Data In 5;
                                 .D[6]:=TIID^Device 1 (EtherCAT)^Term 1 (EK1200)^Term 2 (EK1122)^Hoffman Box Vac EK1 (EK1100)^E5 (EL6022)^COM Inputs Channel 1^Data In 6;
                                 .D[7]:=TIID^Device 1 (EtherCAT)^Term 1 (EK1200)^Term 2 (EK1122)^Hoffman Box Vac EK1 (EK1100)^E5 (EL6022)^COM Inputs Channel 1^Data In 7;
                                 .D[8]:=TIID^Device 1 (EtherCAT)^Term 1 (EK1200)^Term 2 (EK1122)^Hoffman Box Vac EK1 (EK1100)^E5 (EL6022)^COM Inputs Channel 1^Data In 8;
                                 .D[9]:=TIID^Device 1 (EtherCAT)^Term 1 (EK1200)^Term 2 (EK1122)^Hoffman Box Vac EK1 (EK1100)^E5 (EL6022)^COM Inputs Channel 1^Data In 9;
                                 .D[10]:=TIID^Device 1 (EtherCAT)^Term 1 (EK1200)^Term 2 (EK1122)^Hoffman Box Vac EK1 (EK1100)^E5 (EL6022)^COM Inputs Channel 1^Data In 10;
                                 .D[11]:=TIID^Device 1 (EtherCAT)^Term 1 (EK1200)^Term 2 (EK1122)^Hoffman Box Vac EK1 (EK1100)^E5 (EL6022)^COM Inputs Channel 1^Data In 11;
                                 .D[12]:=TIID^Device 1 (EtherCAT)^Term 1 (EK1200)^Term 2 (EK1122)^Hoffman Box Vac EK1 (EK1100)^E5 (EL6022)^COM Inputs Channel 1^Data In 12;
                                 .D[13]:=TIID^Device 1 (EtherCAT)^Term 1 (EK1200)^Term 2 (EK1122)^Hoffman Box Vac EK1 (EK1100)^E5 (EL6022)^COM Inputs Channel 1^Data In 13;
                                 .D[14]:=TIID^Device 1 (EtherCAT)^Term 1 (EK1200)^Term 2 (EK1122)^Hoffman Box Vac EK1 (EK1100)^E5 (EL6022)^COM Inputs Channel 1^Data In 14;
                                 .D[15]:=TIID^Device 1 (EtherCAT)^Term 1 (EK1200)^Term 2 (EK1122)^Hoffman Box Vac EK1 (EK1100)^E5 (EL6022)^COM Inputs Channel 1^Data In 15;
                                 .D[16]:=TIID^Device 1 (EtherCAT)^Term 1 (EK1200)^Term 2 (EK1122)^Hoffman Box Vac EK1 (EK1100)^E5 (EL6022)^COM Inputs Channel 1^Data In 16;
                                 .D[17]:=TIID^Device 1 (EtherCAT)^Term 1 (EK1200)^Term 2 (EK1122)^Hoffman Box Vac EK1 (EK1100)^E5 (EL6022)^COM Inputs Channel 1^Data In 17;
                                 .D[18]:=TIID^Device 1 (EtherCAT)^Term 1 (EK1200)^Term 2 (EK1122)^Hoffman Box Vac EK1 (EK1100)^E5 (EL6022)^COM Inputs Channel 1^Data In 18;
                                 .D[19]:=TIID^Device 1 (EtherCAT)^Term 1 (EK1200)^Term 2 (EK1122)^Hoffman Box Vac EK1 (EK1100)^E5 (EL6022)^COM Inputs Channel 1^Data In 19;
                                 .D[20]:=TIID^Device 1 (EtherCAT)^Term 1 (EK1200)^Term 2 (EK1122)^Hoffman Box Vac EK1 (EK1100)^E5 (EL6022)^COM Inputs Channel 1^Data In 20;
                                 .D[21]:=TIID^Device 1 (EtherCAT)^Term 1 (EK1200)^Term 2 (EK1122)^Hoffman Box Vac EK1 (EK1100)^E5 (EL6022)^COM Inputs Channel 1^Data In 21
    '}
    K2S17_E5_CH1_stComIn		AT %I*	:	EL6inData22B;
    {attribute	'TcLinkTo'	:=	'.Ctrl:=TIID^Device 1 (EtherCAT)^Term 1 (EK1200)^Term 2 (EK1122)^Hoffman Box Vac EK1 (EK1100)^E5 (EL6022)^COM Outputs Channel 1^Ctrl;
                                 .D[0]:=TIID^Device 1 (EtherCAT)^Term 1 (EK1200)^Term 2 (EK1122)^Hoffman Box Vac EK1 (EK1100)^E5 (EL6022)^COM Outputs Channel 1^Data Out 0;
                                 .D[1]:=TIID^Device 1 (EtherCAT)^Term 1 (EK1200)^Term 2 (EK1122)^Hoffman Box Vac EK1 (EK1100)^E5 (EL6022)^COM Outputs Channel 1^Data Out 1;
                                 .D[2]:=TIID^Device 1 (EtherCAT)^Term 1 (EK1200)^Term 2 (EK1122)^Hoffman Box Vac EK1 (EK1100)^E5 (EL6022)^COM Outputs Channel 1^Data Out 2;
                                 .D[3]:=TIID^Device 1 (EtherCAT)^Term 1 (EK1200)^Term 2 (EK1122)^Hoffman Box Vac EK1 (EK1100)^E5 (EL6022)^COM Outputs Channel 1^Data Out 3;
                                 .D[4]:=TIID^Device 1 (EtherCAT)^Term 1 (EK1200)^Term 2 (EK1122)^Hoffman Box Vac EK1 (EK1100)^E5 (EL6022)^COM Outputs Channel 1^Data Out 4;
                                 .D[5]:=TIID^Device 1 (EtherCAT)^Term 1 (EK1200)^Term 2 (EK1122)^Hoffman Box Vac EK1 (EK1100)^E5 (EL6022)^COM Outputs Channel 1^Data Out 5;
                                 .D[6]:=TIID^Device 1 (EtherCAT)^Term 1 (EK1200)^Term 2 (EK1122)^Hoffman Box Vac EK1 (EK1100)^E5 (EL6022)^COM Outputs Channel 1^Data Out 6;
                                 .D[7]:=TIID^Device 1 (EtherCAT)^Term 1 (EK1200)^Term 2 (EK1122)^Hoffman Box Vac EK1 (EK1100)^E5 (EL6022)^COM Outputs Channel 1^Data Out 7;
                                 .D[8]:=TIID^Device 1 (EtherCAT)^Term 1 (EK1200)^Term 2 (EK1122)^Hoffman Box Vac EK1 (EK1100)^E5 (EL6022)^COM Outputs Channel 1^Data Out 8;
                                 .D[9]:=TIID^Device 1 (EtherCAT)^Term 1 (EK1200)^Term 2 (EK1122)^Hoffman Box Vac EK1 (EK1100)^E5 (EL6022)^COM Outputs Channel 1^Data Out 9;
                                 .D[10]:=TIID^Device 1 (EtherCAT)^Term 1 (EK1200)^Term 2 (EK1122)^Hoffman Box Vac EK1 (EK1100)^E5 (EL6022)^COM Outputs Channel 1^Data Out 10;
                                 .D[11]:=TIID^Device 1 (EtherCAT)^Term 1 (EK1200)^Term 2 (EK1122)^Hoffman Box Vac EK1 (EK1100)^E5 (EL6022)^COM Outputs Channel 1^Data Out 11;
                                 .D[12]:=TIID^Device 1 (EtherCAT)^Term 1 (EK1200)^Term 2 (EK1122)^Hoffman Box Vac EK1 (EK1100)^E5 (EL6022)^COM Outputs Channel 1^Data Out 12;
                                 .D[13]:=TIID^Device 1 (EtherCAT)^Term 1 (EK1200)^Term 2 (EK1122)^Hoffman Box Vac EK1 (EK1100)^E5 (EL6022)^COM Outputs Channel 1^Data Out 13;
                                 .D[14]:=TIID^Device 1 (EtherCAT)^Term 1 (EK1200)^Term 2 (EK1122)^Hoffman Box Vac EK1 (EK1100)^E5 (EL6022)^COM Outputs Channel 1^Data Out 14;
                                 .D[15]:=TIID^Device 1 (EtherCAT)^Term 1 (EK1200)^Term 2 (EK1122)^Hoffman Box Vac EK1 (EK1100)^E5 (EL6022)^COM Outputs Channel 1^Data Out 15;
                                 .D[16]:=TIID^Device 1 (EtherCAT)^Term 1 (EK1200)^Term 2 (EK1122)^Hoffman Box Vac EK1 (EK1100)^E5 (EL6022)^COM Outputs Channel 1^Data Out 16;
                                 .D[17]:=TIID^Device 1 (EtherCAT)^Term 1 (EK1200)^Term 2 (EK1122)^Hoffman Box Vac EK1 (EK1100)^E5 (EL6022)^COM Outputs Channel 1^Data Out 17;
                                 .D[18]:=TIID^Device 1 (EtherCAT)^Term 1 (EK1200)^Term 2 (EK1122)^Hoffman Box Vac EK1 (EK1100)^E5 (EL6022)^COM Outputs Channel 1^Data Out 18;
                                 .D[19]:=TIID^Device 1 (EtherCAT)^Term 1 (EK1200)^Term 2 (EK1122)^Hoffman Box Vac EK1 (EK1100)^E5 (EL6022)^COM Outputs Channel 1^Data Out 19;
                                 .D[20]:=TIID^Device 1 (EtherCAT)^Term 1 (EK1200)^Term 2 (EK1122)^Hoffman Box Vac EK1 (EK1100)^E5 (EL6022)^COM Outputs Channel 1^Data Out 20;
                                 .D[21]:=TIID^Device 1 (EtherCAT)^Term 1 (EK1200)^Term 2 (EK1122)^Hoffman Box Vac EK1 (EK1100)^E5 (EL6022)^COM Outputs Channel 1^Data Out 21
    '}
    K2S17_E5_CH1_stComOut		AT %Q*	:	EL6outData22B;

    // SVLS PTM-01
    CRIX_SVLS_SerialRXBuffer : ComBuffer;
    CRIX_SVLS_SerialTXBuffer : ComBuffer;

    // Serial Terminal
    CRIX_SVLS_fbSerialLineControl: SerialLineControl;

    //SERIAL IO CRIX SVLS E4 (EL6021)
    {attribute	'TcLinkTo'	:=	'.Status:=TIID^Device 1 (EtherCAT)^Term 1 (EK1200)^Term 2 (EK1122)^Hoffman Box Vac EK1 (EK1100)^Term 145 (EK1122)^SVLS_PR01 E0 (EK1100)^SVLS_PR01 E4 (EL6021)^COM TxPDO-Map Inputs^Status;
                                 .D[0]:=TIID^Device 1 (EtherCAT)^Term 1 (EK1200)^Term 2 (EK1122)^Hoffman Box Vac EK1 (EK1100)^Term 145 (EK1122)^SVLS_PR01 E0 (EK1100)^SVLS_PR01 E4 (EL6021)^COM TxPDO-Map Inputs^Data In 0;
                                 .D[1]:=TIID^Device 1 (EtherCAT)^Term 1 (EK1200)^Term 2 (EK1122)^Hoffman Box Vac EK1 (EK1100)^Term 145 (EK1122)^SVLS_PR01 E0 (EK1100)^SVLS_PR01 E4 (EL6021)^COM TxPDO-Map Inputs^Data In 1;
                                 .D[2]:=TIID^Device 1 (EtherCAT)^Term 1 (EK1200)^Term 2 (EK1122)^Hoffman Box Vac EK1 (EK1100)^Term 145 (EK1122)^SVLS_PR01 E0 (EK1100)^SVLS_PR01 E4 (EL6021)^COM TxPDO-Map Inputs^Data In 2;
                                 .D[3]:=TIID^Device 1 (EtherCAT)^Term 1 (EK1200)^Term 2 (EK1122)^Hoffman Box Vac EK1 (EK1100)^Term 145 (EK1122)^SVLS_PR01 E0 (EK1100)^SVLS_PR01 E4 (EL6021)^COM TxPDO-Map Inputs^Data In 3;
                                 .D[4]:=TIID^Device 1 (EtherCAT)^Term 1 (EK1200)^Term 2 (EK1122)^Hoffman Box Vac EK1 (EK1100)^Term 145 (EK1122)^SVLS_PR01 E0 (EK1100)^SVLS_PR01 E4 (EL6021)^COM TxPDO-Map Inputs^Data In 4;
                                 .D[5]:=TIID^Device 1 (EtherCAT)^Term 1 (EK1200)^Term 2 (EK1122)^Hoffman Box Vac EK1 (EK1100)^Term 145 (EK1122)^SVLS_PR01 E0 (EK1100)^SVLS_PR01 E4 (EL6021)^COM TxPDO-Map Inputs^Data In 5;
                                 .D[6]:=TIID^Device 1 (EtherCAT)^Term 1 (EK1200)^Term 2 (EK1122)^Hoffman Box Vac EK1 (EK1100)^Term 145 (EK1122)^SVLS_PR01 E0 (EK1100)^SVLS_PR01 E4 (EL6021)^COM TxPDO-Map Inputs^Data In 6;
                                 .D[7]:=TIID^Device 1 (EtherCAT)^Term 1 (EK1200)^Term 2 (EK1122)^Hoffman Box Vac EK1 (EK1100)^Term 145 (EK1122)^SVLS_PR01 E0 (EK1100)^SVLS_PR01 E4 (EL6021)^COM TxPDO-Map Inputs^Data In 7;
                                 .D[8]:=TIID^Device 1 (EtherCAT)^Term 1 (EK1200)^Term 2 (EK1122)^Hoffman Box Vac EK1 (EK1100)^Term 145 (EK1122)^SVLS_PR01 E0 (EK1100)^SVLS_PR01 E4 (EL6021)^COM TxPDO-Map Inputs^Data In 8;
                                 .D[9]:=TIID^Device 1 (EtherCAT)^Term 1 (EK1200)^Term 2 (EK1122)^Hoffman Box Vac EK1 (EK1100)^Term 145 (EK1122)^SVLS_PR01 E0 (EK1100)^SVLS_PR01 E4 (EL6021)^COM TxPDO-Map Inputs^Data In 9;
                                 .D[10]:=TIID^Device 1 (EtherCAT)^Term 1 (EK1200)^Term 2 (EK1122)^Hoffman Box Vac EK1 (EK1100)^Term 145 (EK1122)^SVLS_PR01 E0 (EK1100)^SVLS_PR01 E4 (EL6021)^COM TxPDO-Map Inputs^Data In 10;
                                 .D[11]:=TIID^Device 1 (EtherCAT)^Term 1 (EK1200)^Term 2 (EK1122)^Hoffman Box Vac EK1 (EK1100)^Term 145 (EK1122)^SVLS_PR01 E0 (EK1100)^SVLS_PR01 E4 (EL6021)^COM TxPDO-Map Inputs^Data In 11;
                                 .D[12]:=TIID^Device 1 (EtherCAT)^Term 1 (EK1200)^Term 2 (EK1122)^Hoffman Box Vac EK1 (EK1100)^Term 145 (EK1122)^SVLS_PR01 E0 (EK1100)^SVLS_PR01 E4 (EL6021)^COM TxPDO-Map Inputs^Data In 12;
                                 .D[13]:=TIID^Device 1 (EtherCAT)^Term 1 (EK1200)^Term 2 (EK1122)^Hoffman Box Vac EK1 (EK1100)^Term 145 (EK1122)^SVLS_PR01 E0 (EK1100)^SVLS_PR01 E4 (EL6021)^COM TxPDO-Map Inputs^Data In 13;
                                 .D[14]:=TIID^Device 1 (EtherCAT)^Term 1 (EK1200)^Term 2 (EK1122)^Hoffman Box Vac EK1 (EK1100)^Term 145 (EK1122)^SVLS_PR01 E0 (EK1100)^SVLS_PR01 E4 (EL6021)^COM TxPDO-Map Inputs^Data In 14;
                                 .D[15]:=TIID^Device 1 (EtherCAT)^Term 1 (EK1200)^Term 2 (EK1122)^Hoffman Box Vac EK1 (EK1100)^Term 145 (EK1122)^SVLS_PR01 E0 (EK1100)^SVLS_PR01 E4 (EL6021)^COM TxPDO-Map Inputs^Data In 15;
                                 .D[16]:=TIID^Device 1 (EtherCAT)^Term 1 (EK1200)^Term 2 (EK1122)^Hoffman Box Vac EK1 (EK1100)^Term 145 (EK1122)^SVLS_PR01 E0 (EK1100)^SVLS_PR01 E4 (EL6021)^COM TxPDO-Map Inputs^Data In 16;
                                 .D[17]:=TIID^Device 1 (EtherCAT)^Term 1 (EK1200)^Term 2 (EK1122)^Hoffman Box Vac EK1 (EK1100)^Term 145 (EK1122)^SVLS_PR01 E0 (EK1100)^SVLS_PR01 E4 (EL6021)^COM TxPDO-Map Inputs^Data In 17;
                                 .D[18]:=TIID^Device 1 (EtherCAT)^Term 1 (EK1200)^Term 2 (EK1122)^Hoffman Box Vac EK1 (EK1100)^Term 145 (EK1122)^SVLS_PR01 E0 (EK1100)^SVLS_PR01 E4 (EL6021)^COM TxPDO-Map Inputs^Data In 18;
                                 .D[19]:=TIID^Device 1 (EtherCAT)^Term 1 (EK1200)^Term 2 (EK1122)^Hoffman Box Vac EK1 (EK1100)^Term 145 (EK1122)^SVLS_PR01 E0 (EK1100)^SVLS_PR01 E4 (EL6021)^COM TxPDO-Map Inputs^Data In 19;
                                 .D[20]:=TIID^Device 1 (EtherCAT)^Term 1 (EK1200)^Term 2 (EK1122)^Hoffman Box Vac EK1 (EK1100)^Term 145 (EK1122)^SVLS_PR01 E0 (EK1100)^SVLS_PR01 E4 (EL6021)^COM TxPDO-Map Inputs^Data In 20;
                                 .D[21]:=TIID^Device 1 (EtherCAT)^Term 1 (EK1200)^Term 2 (EK1122)^Hoffman Box Vac EK1 (EK1100)^Term 145 (EK1122)^SVLS_PR01 E0 (EK1100)^SVLS_PR01 E4 (EL6021)^COM TxPDO-Map Inputs^Data In 21
    '}
    CRIX_SVLS_stComIn		AT %I*	:	EL6inData22B;
    {attribute	'TcLinkTo'	:=	'.Ctrl:=TIID^Device 1 (EtherCAT)^Term 1 (EK1200)^Term 2 (EK1122)^Hoffman Box Vac EK1 (EK1100)^Term 145 (EK1122)^SVLS_PR01 E0 (EK1100)^SVLS_PR01 E4 (EL6021)^COM RxPDO-Map Outputs^Ctrl;
                                 .D[0]:=TIID^Device 1 (EtherCAT)^Term 1 (EK1200)^Term 2 (EK1122)^Hoffman Box Vac EK1 (EK1100)^Term 145 (EK1122)^SVLS_PR01 E0 (EK1100)^SVLS_PR01 E4 (EL6021)^COM RxPDO-Map Outputs^Data Out 0;
                                 .D[1]:=TIID^Device 1 (EtherCAT)^Term 1 (EK1200)^Term 2 (EK1122)^Hoffman Box Vac EK1 (EK1100)^Term 145 (EK1122)^SVLS_PR01 E0 (EK1100)^SVLS_PR01 E4 (EL6021)^COM RxPDO-Map Outputs^Data Out 1;
                                 .D[2]:=TIID^Device 1 (EtherCAT)^Term 1 (EK1200)^Term 2 (EK1122)^Hoffman Box Vac EK1 (EK1100)^Term 145 (EK1122)^SVLS_PR01 E0 (EK1100)^SVLS_PR01 E4 (EL6021)^COM RxPDO-Map Outputs^Data Out 2;
                                 .D[3]:=TIID^Device 1 (EtherCAT)^Term 1 (EK1200)^Term 2 (EK1122)^Hoffman Box Vac EK1 (EK1100)^Term 145 (EK1122)^SVLS_PR01 E0 (EK1100)^SVLS_PR01 E4 (EL6021)^COM RxPDO-Map Outputs^Data Out 3;
                                 .D[4]:=TIID^Device 1 (EtherCAT)^Term 1 (EK1200)^Term 2 (EK1122)^Hoffman Box Vac EK1 (EK1100)^Term 145 (EK1122)^SVLS_PR01 E0 (EK1100)^SVLS_PR01 E4 (EL6021)^COM RxPDO-Map Outputs^Data Out 4;
                                 .D[5]:=TIID^Device 1 (EtherCAT)^Term 1 (EK1200)^Term 2 (EK1122)^Hoffman Box Vac EK1 (EK1100)^Term 145 (EK1122)^SVLS_PR01 E0 (EK1100)^SVLS_PR01 E4 (EL6021)^COM RxPDO-Map Outputs^Data Out 5;
                                 .D[6]:=TIID^Device 1 (EtherCAT)^Term 1 (EK1200)^Term 2 (EK1122)^Hoffman Box Vac EK1 (EK1100)^Term 145 (EK1122)^SVLS_PR01 E0 (EK1100)^SVLS_PR01 E4 (EL6021)^COM RxPDO-Map Outputs^Data Out 6;
                                 .D[7]:=TIID^Device 1 (EtherCAT)^Term 1 (EK1200)^Term 2 (EK1122)^Hoffman Box Vac EK1 (EK1100)^Term 145 (EK1122)^SVLS_PR01 E0 (EK1100)^SVLS_PR01 E4 (EL6021)^COM RxPDO-Map Outputs^Data Out 7;
                                 .D[8]:=TIID^Device 1 (EtherCAT)^Term 1 (EK1200)^Term 2 (EK1122)^Hoffman Box Vac EK1 (EK1100)^Term 145 (EK1122)^SVLS_PR01 E0 (EK1100)^SVLS_PR01 E4 (EL6021)^COM RxPDO-Map Outputs^Data Out 8;
                                 .D[9]:=TIID^Device 1 (EtherCAT)^Term 1 (EK1200)^Term 2 (EK1122)^Hoffman Box Vac EK1 (EK1100)^Term 145 (EK1122)^SVLS_PR01 E0 (EK1100)^SVLS_PR01 E4 (EL6021)^COM RxPDO-Map Outputs^Data Out 9;
                                 .D[10]:=TIID^Device 1 (EtherCAT)^Term 1 (EK1200)^Term 2 (EK1122)^Hoffman Box Vac EK1 (EK1100)^Term 145 (EK1122)^SVLS_PR01 E0 (EK1100)^SVLS_PR01 E4 (EL6021)^COM RxPDO-Map Outputs^Data Out 10;
                                 .D[11]:=TIID^Device 1 (EtherCAT)^Term 1 (EK1200)^Term 2 (EK1122)^Hoffman Box Vac EK1 (EK1100)^Term 145 (EK1122)^SVLS_PR01 E0 (EK1100)^SVLS_PR01 E4 (EL6021)^COM RxPDO-Map Outputs^Data Out 11;
                                 .D[12]:=TIID^Device 1 (EtherCAT)^Term 1 (EK1200)^Term 2 (EK1122)^Hoffman Box Vac EK1 (EK1100)^Term 145 (EK1122)^SVLS_PR01 E0 (EK1100)^SVLS_PR01 E4 (EL6021)^COM RxPDO-Map Outputs^Data Out 12;
                                 .D[13]:=TIID^Device 1 (EtherCAT)^Term 1 (EK1200)^Term 2 (EK1122)^Hoffman Box Vac EK1 (EK1100)^Term 145 (EK1122)^SVLS_PR01 E0 (EK1100)^SVLS_PR01 E4 (EL6021)^COM RxPDO-Map Outputs^Data Out 13;
                                 .D[14]:=TIID^Device 1 (EtherCAT)^Term 1 (EK1200)^Term 2 (EK1122)^Hoffman Box Vac EK1 (EK1100)^Term 145 (EK1122)^SVLS_PR01 E0 (EK1100)^SVLS_PR01 E4 (EL6021)^COM RxPDO-Map Outputs^Data Out 14;
                                 .D[15]:=TIID^Device 1 (EtherCAT)^Term 1 (EK1200)^Term 2 (EK1122)^Hoffman Box Vac EK1 (EK1100)^Term 145 (EK1122)^SVLS_PR01 E0 (EK1100)^SVLS_PR01 E4 (EL6021)^COM RxPDO-Map Outputs^Data Out 15;
                                 .D[16]:=TIID^Device 1 (EtherCAT)^Term 1 (EK1200)^Term 2 (EK1122)^Hoffman Box Vac EK1 (EK1100)^Term 145 (EK1122)^SVLS_PR01 E0 (EK1100)^SVLS_PR01 E4 (EL6021)^COM RxPDO-Map Outputs^Data Out 16;
                                 .D[17]:=TIID^Device 1 (EtherCAT)^Term 1 (EK1200)^Term 2 (EK1122)^Hoffman Box Vac EK1 (EK1100)^Term 145 (EK1122)^SVLS_PR01 E0 (EK1100)^SVLS_PR01 E4 (EL6021)^COM RxPDO-Map Outputs^Data Out 17;
                                 .D[18]:=TIID^Device 1 (EtherCAT)^Term 1 (EK1200)^Term 2 (EK1122)^Hoffman Box Vac EK1 (EK1100)^Term 145 (EK1122)^SVLS_PR01 E0 (EK1100)^SVLS_PR01 E4 (EL6021)^COM RxPDO-Map Outputs^Data Out 18;
                                 .D[19]:=TIID^Device 1 (EtherCAT)^Term 1 (EK1200)^Term 2 (EK1122)^Hoffman Box Vac EK1 (EK1100)^Term 145 (EK1122)^SVLS_PR01 E0 (EK1100)^SVLS_PR01 E4 (EL6021)^COM RxPDO-Map Outputs^Data Out 19;
                                 .D[20]:=TIID^Device 1 (EtherCAT)^Term 1 (EK1200)^Term 2 (EK1122)^Hoffman Box Vac EK1 (EK1100)^Term 145 (EK1122)^SVLS_PR01 E0 (EK1100)^SVLS_PR01 E4 (EL6021)^COM RxPDO-Map Outputs^Data Out 20;
                                 .D[21]:=TIID^Device 1 (EtherCAT)^Term 1 (EK1200)^Term 2 (EK1122)^Hoffman Box Vac EK1 (EK1100)^Term 145 (EK1122)^SVLS_PR01 E0 (EK1100)^SVLS_PR01 E4 (EL6021)^COM RxPDO-Map Outputs^Data Out 21
    '}
    CRIX_SVLS_stComOut		AT %Q*	:	EL6outData22B;


END_VAR

// ---- GVLs/GVL_COM_VLS.TcGVL
//{attribute 'qualified_only'}
VAR_GLOBAL
    // Define COM Ports/Buffers incl. library Tc2_SerialCom
    VLS_EP1_CH1_SerialRXBuffer : ComBuffer;
    VLS_EP1_CH1_SerialTXBuffer : ComBuffer;

    // Serial Terminal
    VLS_EP1_CH1_fbSerialLineControl: SerialLineControl;

    //SERIAL IO
        {attribute	'TcLinkTo'	:=	'.Status:=TIIB[VLS_EP1 (EP6002-0002)]^COM TxPDO-Map Inputs Channel 1^Status;
                                 .D[0]:=TIIB[VLS_EP1 (EP6002-0002)]^COM TxPDO-Map Inputs Channel 1^Data In 0;
                                 .D[1]:=TIIB[VLS_EP1 (EP6002-0002)]^COM TxPDO-Map Inputs Channel 1^Data In 1;
                                 .D[2]:=TIIB[VLS_EP1 (EP6002-0002)]^COM TxPDO-Map Inputs Channel 1^Data In 2;
                                 .D[3]:=TIIB[VLS_EP1 (EP6002-0002)]^COM TxPDO-Map Inputs Channel 1^Data In 3;
                                 .D[4]:=TIIB[VLS_EP1 (EP6002-0002)]^COM TxPDO-Map Inputs Channel 1^Data In 4;
                                 .D[5]:=TIIB[VLS_EP1 (EP6002-0002)]^COM TxPDO-Map Inputs Channel 1^Data In 5;
                                 .D[6]:=TIIB[VLS_EP1 (EP6002-0002)]^COM TxPDO-Map Inputs Channel 1^Data In 6;
                                 .D[7]:=TIIB[VLS_EP1 (EP6002-0002)]^COM TxPDO-Map Inputs Channel 1^Data In 7;
                                 .D[8]:=TIIB[VLS_EP1 (EP6002-0002)]^COM TxPDO-Map Inputs Channel 1^Data In 8;
                                 .D[9]:=TIIB[VLS_EP1 (EP6002-0002)]^COM TxPDO-Map Inputs Channel 1^Data In 9;
                                 .D[10]:=TIIB[VLS_EP1 (EP6002-0002)]^COM TxPDO-Map Inputs Channel 1^Data In 10;
                                 .D[11]:=TIIB[VLS_EP1 (EP6002-0002)]^COM TxPDO-Map Inputs Channel 1^Data In 11;
                                 .D[12]:=TIIB[VLS_EP1 (EP6002-0002)]^COM TxPDO-Map Inputs Channel 1^Data In 12;
                                 .D[13]:=TIIB[VLS_EP1 (EP6002-0002)]^COM TxPDO-Map Inputs Channel 1^Data In 13;
                                 .D[14]:=TIIB[VLS_EP1 (EP6002-0002)]^COM TxPDO-Map Inputs Channel 1^Data In 14;
                                 .D[15]:=TIIB[VLS_EP1 (EP6002-0002)]^COM TxPDO-Map Inputs Channel 1^Data In 15;
                                 .D[16]:=TIIB[VLS_EP1 (EP6002-0002)]^COM TxPDO-Map Inputs Channel 1^Data In 16;
                                 .D[17]:=TIIB[VLS_EP1 (EP6002-0002)]^COM TxPDO-Map Inputs Channel 1^Data In 17;
                                 .D[18]:=TIIB[VLS_EP1 (EP6002-0002)]^COM TxPDO-Map Inputs Channel 1^Data In 18;
                                 .D[19]:=TIIB[VLS_EP1 (EP6002-0002)]^COM TxPDO-Map Inputs Channel 1^Data In 19;
                                 .D[20]:=TIIB[VLS_EP1 (EP6002-0002)]^COM TxPDO-Map Inputs Channel 1^Data In 20;
                                 .D[21]:=TIIB[VLS_EP1 (EP6002-0002)]^COM TxPDO-Map Inputs Channel 1^Data In 21
    '}
    VLS_EP1_CH1_stComIn			AT %I*	:	EL6inData22B;

    {attribute	'TcLinkTo'	:=	'.Ctrl:=TIIB[VLS_EP1 (EP6002-0002)]^COM RxPDO-Map Outputs Channel 1^Ctrl;
                                 .D[0]:=TIIB[VLS_EP1 (EP6002-0002)]^COM RxPDO-Map Outputs Channel 1^Data Out 0;
                                 .D[1]:=TIIB[VLS_EP1 (EP6002-0002)]^COM RxPDO-Map Outputs Channel 1^Data Out 1;
                                 .D[2]:=TIIB[VLS_EP1 (EP6002-0002)]^COM RxPDO-Map Outputs Channel 1^Data Out 2;
                                 .D[3]:=TIIB[VLS_EP1 (EP6002-0002)]^COM RxPDO-Map Outputs Channel 1^Data Out 3;
                                 .D[4]:=TIIB[VLS_EP1 (EP6002-0002)]^COM RxPDO-Map Outputs Channel 1^Data Out 4;
                                 .D[5]:=TIIB[VLS_EP1 (EP6002-0002)]^COM RxPDO-Map Outputs Channel 1^Data Out 5;
                                 .D[6]:=TIIB[VLS_EP1 (EP6002-0002)]^COM RxPDO-Map Outputs Channel 1^Data Out 6;
                                 .D[7]:=TIIB[VLS_EP1 (EP6002-0002)]^COM RxPDO-Map Outputs Channel 1^Data Out 7;
                                 .D[8]:=TIIB[VLS_EP1 (EP6002-0002)]^COM RxPDO-Map Outputs Channel 1^Data Out 8;
                                 .D[9]:=TIIB[VLS_EP1 (EP6002-0002)]^COM RxPDO-Map Outputs Channel 1^Data Out 9;
                                 .D[10]:=TIIB[VLS_EP1 (EP6002-0002)]^COM RxPDO-Map Outputs Channel 1^Data Out 10;
                                 .D[11]:=TIIB[VLS_EP1 (EP6002-0002)]^COM RxPDO-Map Outputs Channel 1^Data Out 11;
                                 .D[12]:=TIIB[VLS_EP1 (EP6002-0002)]^COM RxPDO-Map Outputs Channel 1^Data Out 12;
                                 .D[13]:=TIIB[VLS_EP1 (EP6002-0002)]^COM RxPDO-Map Outputs Channel 1^Data Out 13;
                                 .D[14]:=TIIB[VLS_EP1 (EP6002-0002)]^COM RxPDO-Map Outputs Channel 1^Data Out 14;
                                 .D[15]:=TIIB[VLS_EP1 (EP6002-0002)]^COM RxPDO-Map Outputs Channel 1^Data Out 15;
                                 .D[16]:=TIIB[VLS_EP1 (EP6002-0002)]^COM RxPDO-Map Outputs Channel 1^Data Out 16;
                                 .D[17]:=TIIB[VLS_EP1 (EP6002-0002)]^COM RxPDO-Map Outputs Channel 1^Data Out 17;
                                 .D[18]:=TIIB[VLS_EP1 (EP6002-0002)]^COM RxPDO-Map Outputs Channel 1^Data Out 18;
                                 .D[19]:=TIIB[VLS_EP1 (EP6002-0002)]^COM RxPDO-Map Outputs Channel 1^Data Out 19;
                                 .D[20]:=TIIB[VLS_EP1 (EP6002-0002)]^COM RxPDO-Map Outputs Channel 1^Data Out 20;
                                 .D[21]:=TIIB[VLS_EP1 (EP6002-0002)]^COM RxPDO-Map Outputs Channel 1^Data Out 21
    '}
    VLS_EP1_CH1_stComOut		AT %Q*	:	EL6outData22B;



END_VAR

// ---- GVLs/GVL_LI3K2.TcGVL
//{attribute 'qualified_only'}
VAR_GLOBAL

    // LI3K2 PTM
    (*
    {attribute 'pytmc' :=' pv: RIX:LI3K2:PTM:01 '}
    {attribute 'TcLinkTo' := '.i_xAtSpd := TIID^Device 1 (EtherCAT)^Term 1 (EK1200)^Term 2 (EK1122)^Mech Room Vac EK1 (EK1101)^Term 45 (EL2794)^Channel 1^Output;
                              .i_xFault := TIID^Device 1 (EtherCAT)^Term 1 (EK1200)^Term 2 (EK1122)^Mech Room Vac EK1 (EK1101)^Term 45 (EL2794)^Channel 2^Output;
                              .q_RunDO := TIID^Device 1 (EtherCAT)^Term 1 (EK1200)^Term 2 (EK1122)^Mech Room Vac EK1 (EK1101)^Term 83 (EL1088)^Channel 1^Input'}
    *)
    // TODO: Update I/O mapping
    RIX_LI3K2_PTM_01 : FB_PTM_TwisTorr;

END_VAR

// ---- GVLs/GVL_Mech_Room.TcGVL
//{attribute 'qualified_only'}
VAR_GLOBAL

    {attribute 'pytmc' :=' pv: CRIXS:MECH:PRO:01 '}
    {attribute 'TcLinkTo' := '.q_xMPStart := TIID^Device 1 (EtherCAT)^Term 1 (EK1200)^Term 2 (EK1122)^Mech Room Vac EK1 (EK1101)^Term 45 (EL2794)^Channel 1^Output;
                              .q_xBPStart := TIID^Device 1 (EtherCAT)^Term 1 (EK1200)^Term 2 (EK1122)^Mech Room Vac EK1 (EK1101)^Term 45 (EL2794)^Channel 2^Output;
                              .i_xMPStatus := TIID^Device 1 (EtherCAT)^Term 1 (EK1200)^Term 2 (EK1122)^Mech Room Vac EK1 (EK1101)^Term 83 (EL1088)^Channel 1^Input;
                              .i_xBPStatus := TIID^Device 1 (EtherCAT)^Term 1 (EK1200)^Term 2 (EK1122)^Mech Room Vac EK1 (EK1101)^Term 83 (EL1088)^Channel 2^Input;
                              .i_xWarning := TIID^Device 1 (EtherCAT)^Term 1 (EK1200)^Term 2 (EK1122)^Mech Room Vac EK1 (EK1101)^Term 83 (EL1088)^Channel 3^Input;
                              .i_xAlarmOK := TIID^Device 1 (EtherCAT)^Term 1 (EK1200)^Term 2 (EK1122)^Mech Room Vac EK1 (EK1101)^Term 83 (EL1088)^Channel 4^Input;
                              .i_xRemote := TIID^Device 1 (EtherCAT)^Term 1 (EK1200)^Term 2 (EK1122)^Mech Room Vac EK1 (EK1101)^Term 83 (EL1088)^Channel 5^Input '}
    MECH_PRO_01 : FB_EbaraDryPump; // ChemRIXS roughing pump in B950-R310 "mechanical room"

    stMECH_PRO_01 : ST_EbaraDryPump;


    {attribute 'pytmc' :=' pv: CRIXS:MECH:VVC:01 '}
    {attribute 'TcLinkTo' := 	'.q_xOPN_DO	:=	TIID^Device 1 (EtherCAT)^Term 1 (EK1200)^Term 2 (EK1122)^Mech Room Vac EK1 (EK1101)^Term 153 (EL2212)^DOX Control Channel 2^Control^Output '}
    MECH_VVC_01 : FB_VVC;

      // Vent valve for rouging line in B950-R310 "mechanical room"

    {attribute 'pytmc' :=' pv: CRIXS:MECH:GPI:01 '}
    {attribute 'TcLinkTo' := 	'.i_iPRESS_R	:=	TIID^Device 1 (EtherCAT)^Term 1 (EK1200)^Term 2 (EK1122)^Mech Room Vac EK1 (EK1101)^Term 92 (EL3174)^AI Standard Channel 1^Value '}
    MECH_GPI_01 : FB_MKS275;   // Guage for rouging line in B950-R310 "mechanical room"

END_VAR

// ---- GVLs/GVL_PLC_Interfaces.TcGVL
//{attribute 'qualified_only'}
VAR_GLOBAL
    (*CRIX Vac*)
    //Outputs
//	fb_ADS_WATCHDOG_VAC_LAMP_TMO:FB_ADS_WATCHDOG;

    (*ETHERCAT BRRIDGE COM STATUS*)
    //0: Other side is in OP state, >0: Error

    {attribute 'pytmc' :=' pv: CRIX:VAC2MOT:ECATBRG:TxPDO_state'}
    {attribute 'TcLinkTo':= 'TIID^Device 1 (EtherCAT)^Term 1 (EK1200)^Term 95 (EL6695)^SYNC Inputs^TxPDO state'}
    xEcatBridge_TxPDO_state AT %I* :BOOL;

    //0: External device connectd, 1: External device not connected
    {attribute 'pytmc' :=' pv: CRIX:VAC2MOT:ECATBRG:External_device_not_connected'}
    {attribute 'TcLinkTo':= 'TIIB[Term 95 (EL6695)]^SYNC Inputs^External device not connected'}
    xEcatBridge_External_device_not_connected AT %I* : BOOL;

    //0 = Data valid, 1 = Data invalid
    {attribute 'pytmc' :=' pv: CRIX:VAC2MOT:ECATBRG:WcState'}
    {attribute 'TcLinkTo' := 'TIID^Device 1 (EtherCAT)^Term 1 (EK1200)^Term 95 (EL6695)^WcState^WcState'}
    xEcatBridge_WcState AT %I* : BOOL;

    (*I/O Inputs to CRIX motion plc*)
    {attribute 'TcLinkTo' :=  'TIID^Device 1 (EtherCAT)^Term 1 (EK1200)^Term 95 (EL6695)^IO Inputs^bMOTY10_IN'}
    xPTC_MOT_Y_10_IN AT %I* : BOOL;

    {attribute 'TcLinkTo' := 'TIID^Device 1 (EtherCAT)^Term 1 (EK1200)^Term 95 (EL6695)^IO Inputs^bMOTY10_OUT'}
    xPTC_MOT_Y_10_OUT AT %I* : BOOL;

    {attribute 'TcLinkTo' :=  'TIID^Device 1 (EtherCAT)^Term 1 (EK1200)^Term 95 (EL6695)^IO Inputs^bMOTY11_IN'}
    xPTC_MOT_Y_11_IN AT %I* : BOOL;

    {attribute 'TcLinkTo' := 'TIID^Device 1 (EtherCAT)^Term 1 (EK1200)^Term 95 (EL6695)^IO Inputs^bMOTY11_OUT'}
    xPTC_MOT_Y_11_OUT AT %I* : BOOL;


    {attribute 'TcLinkTo' :=  'TIID^Device 1 (EtherCAT)^Term 1 (EK1200)^Term 95 (EL6695)^IO Inputs^xSDS_MOT_Z_18_IN
    '}
    xSDS_MOT_Z_18_IN AT %I* : BOOL;

    {attribute 'TcLinkTo' := 'TIID^Device 1 (EtherCAT)^Term 1 (EK1200)^Term 95 (EL6695)^IO Inputs^xSDS_MOT_Z_18_OUT
    '}
    xSDS_MOT_Z_18_OUT AT %I* : BOOL;


    (*I/O Outputs to CRIX Motion PLC*)

    {attribute 'TcLinkTo' :=  'TIID^Device 1 (EtherCAT)^Term 1 (EK1200)^Term 95 (EL6695)^IO Outputs^bCRYO_VGC_01_CLS
    '}
    bCRYO_VGC_01_CLS AT %Q* : BOOL;

    {attribute 'TcLinkTo' :=  'TIID^Device 1 (EtherCAT)^Term 1 (EK1200)^Term 95 (EL6695)^IO Outputs^bCRYO_VGC_01_OPN
    '}
    bCRYO_VGC_01_OPN AT %Q* : BOOL;

    {attribute 'TcLinkTo' :=  'TIID^Device 1 (EtherCAT)^Term 1 (EK1200)^Term 95 (EL6695)^IO Outputs^bCRYO_VGC_02_CLS
    '}
    bCRYO_VGC_02_CLS AT %Q* : BOOL;

    {attribute 'TcLinkTo' :=  'TIID^Device 1 (EtherCAT)^Term 1 (EK1200)^Term 95 (EL6695)^IO Outputs^bCRYO_VGC_02_OPN
    '}
    bCRYO_VGC_02_OPN AT %Q* : BOOL;

    {attribute 'TcLinkTo' :=  'TIID^Device 1 (EtherCAT)^Term 1 (EK1200)^Term 95 (EL6695)^IO Outputs^bSDS_VGC_01_CLS
    '}
    bSDS_VGC_01_CLS AT %Q* : BOOL;

    {attribute 'TcLinkTo' :=  'TIID^Device 1 (EtherCAT)^Term 1 (EK1200)^Term 95 (EL6695)^IO Outputs^bSDS_VGC_01_OPN
    '}
    bSDS_VGC_01_OPN AT %Q* : BOOL;

END_VAR

// ---- GVLs/GVL_PMPS.TcGVL
//{attribute 'qualified_only'}
VAR_GLOBAL
    {attribute 'pytmc' := 'pv: PLC:CRIXS:VAC:FFO:01'}
    {attribute 'TcLinkTo' := '.q_xFastFaultOut:=TIID^Device 1 (EtherCAT)^Term 1 (EK1200)^Term 113 (EK1521-0010)^Term 154 (EK1501-0010)^PMPS_FFO^Channel 1^Output'}
    g_FastFaultOutput1: FB_HardwareFFOutput :=(i_sNetID:='172.21.42.126.1.1');;

    {attribute 'pytmc' := 'pv: PLC:CRIXS:VAC:FFO:02'}
    {attribute 'TcLinkTo' := '.q_xFastFaultOut:=TIID^Device 1 (EtherCAT)^Term 1 (EK1200)^Term 113 (EK1521-0010)^Term 154 (EK1501-0010)^PMPS_PRE^IO Outputs^FFO_Link'}
    g_FastFaultOutput2: FB_HardwareFFOutput :=(i_sNetID:='172.21.42.126.1.1');;


    {attribute 'pytmc' := 'pv: PLC:CRIXS:VAC:ARB:01'}
    fbArbiter1: FB_Arbiter(1);
END_VAR

// ---- GVLs/GVL_Pumps.TcGVL
//{attribute 'qualified_only'}
VAR_GLOBAL

    (* Leybold Pumps *)
    {attribute 'pytmc' :=' pv: CRIXS:TC:PTM:02 '}
    {attribute 'TcLinkTo' := 	'.i_xAtSpd	 :=	TIID^Device 1 (EtherCAT)^Term 1 (EK1200)^Term 2 (EK1122)^Hoffman Box Vac EK1 (EK1100)^E42 (EL1004)^Channel 2^Input;
                                 .i_xFaultNC :=	TIID^Device 1 (EtherCAT)^Term 1 (EK1200)^Term 2 (EK1122)^Hoffman Box Vac EK1 (EK1100)^E42 (EL1004)^Channel 1^Input;
                                 .q_RunDO	 :=	TIID^Device 1 (EtherCAT)^Term 1 (EK1200)^Term 2 (EK1122)^Hoffman Box Vac EK1 (EK1100)^E43 (EL2794)^Channel 3^Output'}
    TC_PTM_02 : FB_PTM_TurboDrive;

    stTC_PTM_02 : ST_LeyboldPTM;

    {attribute 'pytmc' :=' pv: CRIXS:TC:PTM:01 '}
    {attribute 'TcLinkTo' := 	'.i_xAtSpd	 :=	TIID^Device 1 (EtherCAT)^Term 1 (EK1200)^Term 2 (EK1122)^Hoffman Box Vac EK1 (EK1100)^E42 (EL1004)^Channel 4^Input;
                                 .i_xFaultNC :=	TIID^Device 1 (EtherCAT)^Term 1 (EK1200)^Term 2 (EK1122)^Hoffman Box Vac EK1 (EK1100)^E42 (EL1004)^Channel 3^Input;
                                 .q_RunDO	 :=	TIID^Device 1 (EtherCAT)^Term 1 (EK1200)^Term 2 (EK1122)^Hoffman Box Vac EK1 (EK1100)^E43 (EL2794)^Channel 4^Output'}
    TC_PTM_01 : FB_PTM_TurboDrive;

    stTC_PTM_01 : ST_LeyboldPTM;


    (* Pfeiffer Turbo Pumps TC400 *)
    {attribute 'TcLinkTo' := 	'.i_xAtSpd			:=	TIID^Device 1 (EtherCAT)^Term 1 (EK1200)^Term 2 (EK1122)^Hoffman Box Vac EK1 (EK1100)^E46 (EL1004)^Channel 1^Input;
                                 .i_xRemote			:=	TIID^Device 1 (EtherCAT)^Term 1 (EK1200)^Term 2 (EK1122)^Hoffman Box Vac EK1 (EK1100)^E46 (EL1004)^Channel 2^Input;
                                 .i_xFaultNC		:=	TIID^Device 1 (EtherCAT)^Term 1 (EK1200)^Term 2 (EK1122)^Hoffman Box Vac EK1 (EK1100)^E46 (EL1004)^Channel 3^Input;
                                 .q_RunDO			:=	TIID^Device 1 (EtherCAT)^Term 1 (EK1200)^Term 2 (EK1122)^Hoffman Box Vac EK1 (EK1100)^E47 (EL2004)^Channel 1^Output;
                                 .q_xRemote			:=	TIID^Device 1 (EtherCAT)^Term 1 (EK1200)^Term 2 (EK1122)^Hoffman Box Vac EK1 (EK1100)^E47 (EL2004)^Channel 2^Output;
                                 .q_PumpingStation	:=	TIID^Device 1 (EtherCAT)^Term 1 (EK1200)^Term 2 (EK1122)^Hoffman Box Vac EK1 (EK1100)^E47 (EL2004)^Channel 3^Output
    '}
    {attribute 'pytmc' := '
        pv: CRIXS:TC:PTM:03
        io: io
    '}
    TC_PTM_03 : FB_PTM_Pfeiffer;

    stTC_PTM_03 : ST_PfeifferPTM;

    stTC_PTM_03_Pfeiffer_CTRL 	: ARRAY[1..20] OF ST_PfeifferControl;
    stTC_PTM_03_Pfeiffer_RBK 	: ARRAY[1..20] OF ST_PfeifferStatus;

    fbTC_PTM_03_PfeifferCom : FB_PFEIFFER_COM;



    (* Pfeiffer Turbo Pumps TC400 *)

    {attribute 'TcLinkTo' := 	'.i_xAtSpd			:=	TIID^Device 1 (EtherCAT)^Term 1 (EK1200)^Term 2 (EK1122)^Hoffman Box Vac EK1 (EK1100)^E49 (EL1004)^Channel 1^Input;
                                 .i_xRemote			:=	TIID^Device 1 (EtherCAT)^Term 1 (EK1200)^Term 2 (EK1122)^Hoffman Box Vac EK1 (EK1100)^E49 (EL1004)^Channel 2^Input;
                                 .i_xFaultNC		:=	TIID^Device 1 (EtherCAT)^Term 1 (EK1200)^Term 2 (EK1122)^Hoffman Box Vac EK1 (EK1100)^E49 (EL1004)^Channel 3^Input;
                                 .q_RunDO			:=	TIID^Device 1 (EtherCAT)^Term 1 (EK1200)^Term 2 (EK1122)^Hoffman Box Vac EK1 (EK1100)^E50 (EL2004)^Channel 1^Output;
                                 .q_xRemote			:=	TIID^Device 1 (EtherCAT)^Term 1 (EK1200)^Term 2 (EK1122)^Hoffman Box Vac EK1 (EK1100)^E50 (EL2004)^Channel 2^Output;
                                 .q_PumpingStation	:=	TIID^Device 1 (EtherCAT)^Term 1 (EK1200)^Term 2 (EK1122)^Hoffman Box Vac EK1 (EK1100)^E50 (EL2004)^Channel 3^Output
    '}

    {attribute 'pytmc' := '
        pv: CRIXS:SDS:PTM:01
        io: io
    '}
    SDS_PTM_01 : FB_PTM_Pfeiffer;

    stSDS_PTM_01 : ST_PfeifferPTM;  //new

    // Serial port
    stSDS_PTM_01_Pfeiffer_CTRL 	: ARRAY[1..20] OF ST_PfeifferControl;
    stSDS_PTM_01_Pfeiffer_RBK 	: ARRAY[1..20] OF ST_PfeifferStatus;

    fb_SDS_PTM_01_Pfeiffer_PfeifferCom : FB_PFEIFFER_COM;

    (* Pfeiffer Turbo Pumps TC110 *)
    // SVLS

    {attribute 'pytmc' := ' pv: CRIX:SVLS:PTM:01'}
    {attribute 'TcLinkTo' := 	'.i_xAtSpd		      := TIIB[SVLS_PR01 E2 (EL1004)]^Channel 1^Input;
                               .i_xFaultNC		  := TIIB[SVLS_PR01 E2 (EL1004)]^Channel 2^Input;
                               .q_RunDO           := TIIB[SVLS_PR01 E3 (EL2794)]^Channel 1^Output;
                               .q_xReset          := TIIB[SVLS_PR01 E3 (EL2794)]^Channel 2^Output
    '}
    CRIX_SVLS_PTM_01 : FB_PTM_Pfeiffer;
    stCRIX_SVLS_PTM_01 : ST_PfeifferPTM;

    // Serial port
    stCRIX_SVLS_PTM_01_Pfeiffer_CTRL 	: ARRAY[1..20] OF ST_PfeifferControl;
    stCRIX_SVLS_PTM_01_Pfeiffer_RBK 	: ARRAY[1..20] OF ST_PfeifferStatus;

    fb_CRIX_SVLS_PTM_01_PfeifferCom : FB_PFEIFFER_COM;

    // SIP PIP NexTORR Pumps
    {attribute 'pytmc' := ' pv: CRIX:SVLS:PIP:1 '}
    {attribute 'TcLinkTo' := 	'.i_iPRESS		:=	TIIB[SVLS_PR01 E9 (EL3174-0002)]^AI Standard Channel 1^Value;
                                 .i_xIP_ON		:= 	TIIB[SVLS_PR01 E11 (EL1124)]^Channel 1^Input;
                                 .i_xError      :=  TIIB[SVLS_PR01 E11 (EL1124)]^Channel 2^Input;
                                 .q_xHVEna_DO	:= 	TIIB[SVLS_PR01 E3 (EL2794)]^Channel 3^Output
    '}
    CRIX_SVLS_PIP_1 : FB_PIP_SIP;

END_VAR

// ---- GVLs/GVL_Recirculation.TcGVL
//{attribute 'qualified_only'}
VAR_GLOBAL
    (* OverrideMode *)
    {attribute 'pytmc' := 'pv: CRIXS:RCC:VAC:OVRD_MODE'}
    xSystemOverrideMode_RCC	: BOOL := FALSE;

    (* Roughing Manifold Valvese *)

    {attribute 'pytmc' :=' pv: CRIXS:RCC:VRC:01 '}
    {attribute 'TcLinkTo' := 	'.i_xClsLS	:=	TIID^Device 1 (EtherCAT)^Term 1 (EK1200)^Term 2 (EK1122)^Hoffman Box Vac EK1 (EK1100)^VLS_RCC (EK1122)^RCC_EK0 (EK1100)^RCC_E1 (EL1004)^Channel 1^Input;
                                .q_xOPN_DO	:=	TIID^Device 1 (EtherCAT)^Term 1 (EK1200)^Term 2 (EK1122)^Hoffman Box Vac EK1 (EK1100)^VLS_RCC (EK1122)^RCC_EK0 (EK1100)^RCC_E2 (EL2004)^Channel 1^Output'}
    RCC_VRC_01 : FB_VRC_NC_ClsLS;

    (* Roughing Manifold Valvese *)

    {attribute 'pytmc' :=' pv: CRIXS:RCC:VRC:02 '}
    {attribute 'TcLinkTo' := 	'.i_xOpnLS	:=	TIID^Device 1 (EtherCAT)^Term 1 (EK1200)^Term 2 (EK1122)^Hoffman Box Vac EK1 (EK1100)^VLS_RCC (EK1122)^RCC_EK0 (EK1100)^RCC_E1 (EL1004)^Channel 4^Input;
                                 .i_xClsLS	:=	TIID^Device 1 (EtherCAT)^Term 1 (EK1200)^Term 2 (EK1122)^Hoffman Box Vac EK1 (EK1100)^VLS_RCC (EK1122)^RCC_EK0 (EK1100)^RCC_E1 (EL1004)^Channel 2^Input;
                                .q_xOPN_DO	:=	TIID^Device 1 (EtherCAT)^Term 1 (EK1200)^Term 2 (EK1122)^Hoffman Box Vac EK1 (EK1100)^VLS_RCC (EK1122)^RCC_EK0 (EK1100)^RCC_E2 (EL2004)^Channel 2^Output'}
    RCC_VRC_02 : FB_VRC;

    (* Roughing Manifold Valvese *)

    {attribute 'pytmc' :=' pv: CRIXS:RCC:VRC:03 '}
    {attribute 'TcLinkTo' := 	'.i_xClsLS	:=	TIID^Device 1 (EtherCAT)^Term 1 (EK1200)^Term 2 (EK1122)^Hoffman Box Vac EK1 (EK1100)^VLS_RCC (EK1122)^RCC_EK0 (EK1100)^RCC_E1 (EL1004)^Channel 3^Input;
                                .q_xOPN_DO	:=	TIID^Device 1 (EtherCAT)^Term 1 (EK1200)^Term 2 (EK1122)^Hoffman Box Vac EK1 (EK1100)^VLS_RCC (EK1122)^RCC_EK0 (EK1100)^RCC_E2 (EL2004)^Channel 3^Output'}
    RCC_VRC_03 : FB_VRC_NC_ClsLS;

    (* Roughing Manifold Valvese *)

